LIN {X 0,Y 175.973,Z 623.597,A -85,B 0,C 180,E1 -22407.711,E2 -22407.711} C_VEL
LIN {X 0,Y 176.091,Z 624.209,A -85,B 0,C 180,E1 -22410,E2 -22410} C_VEL
LIN {X 0,Y 175.945,Z 624.405,A -85,B 0,C 180,E1 -22414.582,E2 -22414.582} C_VEL
LIN {X 0,Y 176.345,Z 623.273,A -85,B 0,C 180,E1 -22419.173,E2 -22419.173} C_VEL
LIN {X 0,Y 177.477,Z 620.803,A -85,B 0,C 180,E1 -22423.745,E2 -22423.745} C_VEL
LIN {X 0,Y 179.709,Z 616.939,A -85,B 0,C 180,E1 -22428.232,E2 -22428.232} C_VEL
LIN {X 0,Y 182.559,Z 611.727,A -85,B 0,C 180,E1 -22432.493,E2 -22432.493} C_VEL
LIN {X 0,Y 185.735,Z 606.375,A -85,B 0,C 180,E1 -22435.795,E2 -22435.795} C_VEL
LIN {X 0,Y 189.98,Z 599.018,A -85,B 0,C 180,E1 -22439.352,E2 -22439.352} C_VEL
LIN {X 0,Y 194.974,Z 589.893,A -85,B 0,C 180,E1 -22442.731,E2 -22442.731} C_VEL
LIN {X 0,Y 199.815,Z 580.368,A -85,B 0,C 180,E1 -22445.475,E2 -22445.475} C_VEL
LIN {X 0,Y 204.272,Z 570.439,A -85,B 0,C 180,E1 -22447.774,E2 -22447.774} C_VEL
LIN {X 0,Y 208.64,Z 559.5,A -85,B 0,C 180,E1 -22449.793,E2 -22449.793} C_VEL
LIN {X 0,Y 213.078,Z 546.888,A -85,B 0,C 180,E1 -22451.59,E2 -22451.59} C_VEL
LIN {X 0,Y 216.743,Z 534.645,A -85,B 0,C 180,E1 -22452.917,E2 -22452.917} C_VEL
LIN {X 0,Y 219.97,Z 521.133,A -85,B 0,C 180,E1 -22454.02,E2 -22454.02} C_VEL
LIN {X 0,Y 222.451,Z 506.848,A -85,B 0,C 180,E1 -22454.855,E2 -22454.855} C_VEL
LIN {X 0,Y 224.016,Z 492.183,A -85,B 0,C 180,E1 -22455.41,E2 -22455.41} C_VEL
LIN {X 0,Y 227.477,Z 439.874,A -85,B 0,C 180,E1 -22456.878,E2 -22456.878} C_VEL
LIN {X 0,Y 222.194,Z 427.229,A -85,B 0,C 180,E1 -22459.105,E2 -22459.105} C_VEL
LIN {X 0,Y 216.883,Z 416.225,A -85,B 0,C 180,E1 -22461.484,E2 -22461.484} C_VEL
LIN {X 0,Y 210.927,Z 405.095,A -85,B 0,C 180,E1 -22464.409,E2 -22464.409} C_VEL
LIN {X 0,Y 204.85,Z 394.973,A -85,B 0,C 180,E1 -22467.765,E2 -22467.765} C_VEL
LIN {X 0,Y 201.102,Z 389.341,A -85,B 0,C 180,E1 -22470.085,E2 -22470.085} C_VEL
LIN {X 0,Y 197.646,Z 384.334,A -85,B 0,C 180,E1 -22472.467,E2 -22472.467} C_VEL
LIN {X 0,Y 194.879,Z 381.371,A -85,B 0,C 180,E1 -22474.511,E2 -22474.511} C_VEL
LIN {X 0,Y 193.552,Z 379.243,A -85,B 0,C 180,E1 -22475.645,E2 -22475.645} C_VEL
LIN {X 0,Y 190.782,Z 376.698,A -85,B 0,C 180,E1 -22478.065,E2 -22478.065} C_VEL
LIN {X 0,Y 189.1,Z 373.76,A -85,B 0,C 180,E1 -22479.893,E2 -22479.893} C_VEL
LIN {X 0,Y 186.16,Z 371.606,A -85,B 0,C 180,E1 -22483.271,E2 -22483.271} C_VEL
LIN {X 0,Y 184.729,Z 369.094,A -85,B 0,C 180,E1 -22485.543,E2 -22485.543} C_VEL
LIN {X 0,Y 184.415,Z 367.934,A -85,B 0,C 180,E1 -22486.221,E2 -22486.221} C_VEL
LIN {X 0,Y 180.968,Z 365.75,A -85,B 0,C 180,E1 -22497.775,E2 -22497.775} C_VEL
LIN {X 0,Y 181.188,Z 365.794,A -85,B 0,C 180,E1 -22500.556,E2 -22500.556} C_VEL
LIN {X 0,Y 183.53,Z 367.618,A -85,B 0,C 180,E1 -22507.703,E2 -22507.703} C_VEL
LIN {X 0,Y 184.611,Z 368.106,A -85,B 0,C 180,E1 -22509.542,E2 -22509.542} C_VEL
LIN {X 0,Y 185.587,Z 370.744,A -85,B 0,C 180,E1 -22511.33,E2 -22511.33} C_VEL
LIN {X 0,Y 187.715,Z 373.002,A -85,B 0,C 180,E1 -22514.086,E2 -22514.086} C_VEL
LIN {X 0,Y 189.365,Z 373.966,A -85,B 0,C 180,E1 -22515.817,E2 -22515.817} C_VEL
LIN {X 0,Y 191.087,Z 377.097,A -85,B 0,C 180,E1 -22517.669,E2 -22517.669} C_VEL
LIN {X 0,Y 193.934,Z 379.745,A -85,B 0,C 180,E1 -22520.116,E2 -22520.116} C_VEL
LIN {X 0,Y 196.242,Z 383.109,A -85,B 0,C 180,E1 -22521.985,E2 -22521.985} C_VEL
LIN {X 0,Y 198.131,Z 385.043,A -85,B 0,C 180,E1 -22523.323,E2 -22523.323} C_VEL
LIN {X 0,Y 200.929,Z 388.709,A -85,B 0,C 180,E1 -22525.212,E2 -22525.212} C_VEL
LIN {X 0,Y 202.67,Z 391.076,A -85,B 0,C 180,E1 -22526.31,E2 -22526.31} C_VEL
LIN {X 0,Y 205.511,Z 394.828,A -85,B 0,C 180,E1 -22527.98,E2 -22527.98} C_VEL
LIN {X 0,Y 210.882,Z 402.349,A -85,B 0,C 180,E1 -22530.844,E2 -22530.844} C_VEL
LIN {X 0,Y 217.896,Z 413.285,A -85,B 0,C 180,E1 -22534.155,E2 -22534.155} C_VEL
LIN {X 0,Y 222.849,Z 422.031,A -85,B 0,C 180,E1 -22536.28,E2 -22536.28} C_VEL
LIN {X 0,Y 227.882,Z 432.924,A -85,B 0,C 180,E1 -22538.349,E2 -22538.349} C_VEL
LIN {X 0,Y 223.972,Z 490.841,A -85,B 0,C 180,E1 -22540.036,E2 -22540.036} C_VEL
LIN {X 0,Y 222.064,Z 505.188,A -85,B 0,C 180,E1 -22540.748,E2 -22540.748} C_VEL
LIN {X 0,Y 219.175,Z 519.704,A -85,B 0,C 180,E1 -22541.795,E2 -22541.795} C_VEL
LIN {X 0,Y 215.825,Z 532.368,A -85,B 0,C 180,E1 -22543.025,E2 -22543.025} C_VEL
LIN {X 0,Y 212.116,Z 544.319,A -85,B 0,C 180,E1 -22544.573,E2 -22544.573} C_VEL
LIN {X 0,Y 207.881,Z 555.831,A -85,B 0,C 180,E1 -22546.462,E2 -22546.462} C_VEL
LIN {X 0,Y 203.787,Z 565.394,A -85,B 0,C 180,E1 -22548.404,E2 -22548.404} C_VEL
LIN {X 0,Y 199.332,Z 575.034,A -85,B 0,C 180,E1 -22550.867,E2 -22550.867} C_VEL
LIN {X 0,Y 195.109,Z 583.394,A -85,B 0,C 180,E1 -22553.534,E2 -22553.534} C_VEL
LIN {X 0,Y 190.261,Z 591.993,A -85,B 0,C 180,E1 -22556.985,E2 -22556.985} C_VEL
LIN {X 0,Y 186.147,Z 598.901,A -85,B 0,C 180,E1 -22560.605,E2 -22560.605} C_VEL
LIN {X 0,Y 183.235,Z 603.656,A -85,B 0,C 180,E1 -22563.827,E2 -22563.827} C_VEL
LIN {X 0,Y 180.146,Z 608.557,A -85,B 0,C 180,E1 -22568.246,E2 -22568.246} C_VEL
LIN {X 0,Y 178.42,Z 611.225,A -85,B 0,C 180,E1 -22571.632,E2 -22571.632} C_VEL
LIN {X 0,Y 176.763,Z 613.538,A -85,B 0,C 180,E1 -22576.198,E2 -22576.198} C_VEL
LIN {X 0,Y 176.071,Z 614.498,A -85,B 0,C 180,E1 -22580.813,E2 -22580.813} C_VEL
LIN {X 0,Y 175.97,Z 614.139,A -85,B 0,C 180,E1 -22585.418,E2 -22585.418} C_VEL
LIN {X 0,Y 176.17,Z 612.472,A -85,B 0,C 180,E1 -22590,E2 -22590} C_VEL
LIN {X 0,Y 176.9,Z 609.462,A -85,B 0,C 180,E1 -22594.557,E2 -22594.557} C_VEL
LIN {X 0,Y 178.404,Z 605.021,A -85,B 0,C 180,E1 -22599.066,E2 -22599.066} C_VEL
LIN {X 0,Y 180.075,Z 600.613,A -85,B 0,C 180,E1 -22602.395,E2 -22602.395} C_VEL
LIN {X 0,Y 182.054,Z 595.264,A -85,B 0,C 180,E1 -22605.678,E2 -22605.678} C_VEL
LIN {X 0,Y 184.936,Z 587.607,A -85,B 0,C 180,E1 -22609.422,E2 -22609.422} C_VEL
LIN {X 0,Y 188.315,Z 579.592,A -85,B 0,C 180,E1 -22612.491,E2 -22612.491} C_VEL
LIN {X 0,Y 191.947,Z 569.95,A -85,B 0,C 180,E1 -22615.481,E2 -22615.481} C_VEL
LIN {X 0,Y 195.507,Z 559.268,A -85,B 0,C 180,E1 -22618.152,E2 -22618.152} C_VEL
LIN {X 0,Y 198.843,Z 548.7,A -85,B 0,C 180,E1 -22620.242,E2 -22620.242} C_VEL
LIN {X 0,Y 202.027,Z 537.334,A -85,B 0,C 180,E1 -22622.04,E2 -22622.04} C_VEL
LIN {X 0,Y 204.873,Z 525.038,A -85,B 0,C 180,E1 -22623.584,E2 -22623.584} C_VEL
LIN {X 0,Y 207.454,Z 511.398,A -85,B 0,C 180,E1 -22624.868,E2 -22624.868} C_VEL
LIN {X 0,Y 209.362,Z 497.206,A -85,B 0,C 180,E1 -22625.828,E2 -22625.828} C_VEL
LIN {X 0,Y 210.555,Z 483.575,A -85,B 0,C 180,E1 -22626.407,E2 -22626.407} C_VEL
LIN {X 0,Y 214.132,Z 420.681,A -85,B 0,C 180,E1 -22628.327,E2 -22628.327} C_VEL
LIN {X 0,Y 209.725,Z 410.077,A -85,B 0,C 180,E1 -22629.873,E2 -22629.873} C_VEL
LIN {X 0,Y 202.836,Z 397.568,A -85,B 0,C 180,E1 -22632.31,E2 -22632.31} C_VEL
LIN {X 0,Y 195.932,Z 386.643,A -85,B 0,C 180,E1 -22634.959,E2 -22634.959} C_VEL
LIN {X 0,Y 191.272,Z 379.912,A -85,B 0,C 180,E1 -22636.904,E2 -22636.904} C_VEL
LIN {X 0,Y 188.461,Z 376.039,A -85,B 0,C 180,E1 -22638.153,E2 -22638.153} C_VEL
LIN {X 0,Y 185.501,Z 371.965,A -85,B 0,C 180,E1 -22639.547,E2 -22639.547} C_VEL
LIN {X 0,Y 183.117,Z 369.127,A -85,B 0,C 180,E1 -22640.708,E2 -22640.708} C_VEL
LIN {X 0,Y 182.006,Z 367.177,A -85,B 0,C 180,E1 -22641.312,E2 -22641.312} C_VEL
LIN {X 0,Y 179.721,Z 365.124,A -85,B 0,C 180,E1 -22642.472,E2 -22642.472} C_VEL
LIN {X 0,Y 178.594,Z 362.743,A -85,B 0,C 180,E1 -22643.165,E2 -22643.165} C_VEL
LIN {X 0,Y 178.432,Z 361.874,A -85,B 0,C 180,E1 -22643.38,E2 -22643.38} C_VEL
LIN {X 0,Y 178.486,Z 361.865,A -85,B 0,C 180,E1 -22646.546,E2 -22646.546} C_VEL
LIN {X 0,Y 178.441,Z 361.868,A -85,B 0,C 180,E1 -22651.794,E2 -22651.794} C_VEL
LIN {X 0,Y 178.507,Z 361.874,A -85,B 0,C 180,E1 -22654.896,E2 -22654.896} C_VEL
LIN {X 0,Y 178.608,Z 361.83,A -85,B 0,C 180,E1 -22661.651,E2 -22661.651} C_VEL
LIN {X 0,Y 178.636,Z 361.834,A -85,B 0,C 180,E1 -22666.345,E2 -22666.345} C_VEL
LIN {X 0,Y 178.908,Z 361.788,A -85,B 0,C 180,E1 -22670.959,E2 -22670.959} C_VEL
LIN {X 0,Y 179.145,Z 361.792,A -85,B 0,C 180,E1 -22677.751,E2 -22677.751} C_VEL
LIN {X 0,Y 179.348,Z 361.762,A -85,B 0,C 180,E1 -22679.999,E2 -22679.999} C_VEL
LIN {X 0,Y 178.84,Z 361.827,A -85,B 0,C 180,E1 -22684.507,E2 -22684.507} C_VEL
LIN {X 0,Y 178.908,Z 361.819,A -85,B 0,C 180,E1 -22689.04,E2 -22689.04} C_VEL
LIN {X 0,Y 178.661,Z 361.848,A -85,B 0,C 180,E1 -22693.651,E2 -22693.651} C_VEL
LIN {X 0,Y 178.624,Z 361.855,A -85,B 0,C 180,E1 -22699.215,E2 -22699.215} C_VEL
LIN {X 0,Y 178.52,Z 361.869,A -85,B 0,C 180,E1 -22705.113,E2 -22705.113} C_VEL
LIN {X 0,Y 178.464,Z 361.884,A -85,B 0,C 180,E1 -22710.793,E2 -22710.793} C_VEL
LIN {X 0,Y 178.485,Z 361.939,A -85,B 0,C 180,E1 -22711.365,E2 -22711.365} C_VEL
LIN {X 0,Y 179.333,Z 364.467,A -85,B 0,C 180,E1 -22711.941,E2 -22711.941} C_VEL
LIN {X 0,Y 181.332,Z 366.723,A -85,B 0,C 180,E1 -22713,E2 -22713} C_VEL
LIN {X 0,Y 182.467,Z 367.748,A -85,B 0,C 180,E1 -22713.563,E2 -22713.563} C_VEL
LIN {X 0,Y 184.533,Z 370.957,A -85,B 0,C 180,E1 -22714.636,E2 -22714.636} C_VEL
LIN {X 0,Y 186.21,Z 372.706,A -85,B 0,C 180,E1 -22715.418,E2 -22715.418} C_VEL
LIN {X 0,Y 188.828,Z 376.357,A -85,B 0,C 180,E1 -22716.641,E2 -22716.641} C_VEL
LIN {X 0,Y 194.381,Z 385.325,A -85,B 0,C 180,E1 -22719.1,E2 -22719.1} C_VEL
LIN {X 0,Y 201.137,Z 397.747,A -85,B 0,C 180,E1 -22721.848,E2 -22721.848} C_VEL
LIN {X 0,Y 206.577,Z 409.402,A -85,B 0,C 180,E1 -22723.922,E2 -22723.922} C_VEL
LIN {X 0,Y 211.631,Z 421.789,A -85,B 0,C 180,E1 -22725.765,E2 -22725.765} C_VEL
LIN {X 0,Y 213.853,Z 427.885,A -85,B 0,C 180,E1 -22726.56,E2 -22726.56} C_VEL
LIN {X 0,Y 212.024,Z 460.209,A -85,B 0,C 180,E1 -22727.546,E2 -22727.546} C_VEL
LIN {X 0,Y 211.141,Z 466.055,A -85,B 0,C 180,E1 -22727.599,E2 -22727.599} C_VEL
LIN {X 0,Y 205.631,Z 485.05,A -85,B 0,C 180,E1 -22727.161,E2 -22727.161} C_VEL
LIN {X 0,Y 204.839,Z 490.89,A -85,B 0,C 180,E1 -22727.236,E2 -22727.236} C_VEL
LIN {X 0,Y 203.51,Z 505.696,A -85,B 0,C 180,E1 -22727.836,E2 -22727.836} C_VEL
LIN {X 0,Y 201.524,Z 518.899,A -85,B 0,C 180,E1 -22728.667,E2 -22728.667} C_VEL
LIN {X 0,Y 198.648,Z 533.064,A -85,B 0,C 180,E1 -22729.949,E2 -22729.949} C_VEL
LIN {X 0,Y 195.227,Z 546.537,A -85,B 0,C 180,E1 -22731.612,E2 -22731.612} C_VEL
LIN {X 0,Y 191.793,Z 558.043,A -85,B 0,C 180,E1 -22733.454,E2 -22733.454} C_VEL
LIN {X 0,Y 187.889,Z 569.824,A -85,B 0,C 180,E1 -22735.87,E2 -22735.87} C_VEL
LIN {X 0,Y 184.218,Z 579.566,A -85,B 0,C 180,E1 -22738.361,E2 -22738.361} C_VEL
LIN {X 0,Y 180.311,Z 589.317,A -85,B 0,C 180,E1 -22741.48,E2 -22741.48} C_VEL
LIN {X 0,Y 177.019,Z 597.403,A -85,B 0,C 180,E1 -22744.736,E2 -22744.736} C_VEL
LIN {X 0,Y 173.979,Z 605.158,A -85,B 0,C 180,E1 -22748.681,E2 -22748.681} C_VEL
LIN {X 0,Y 171.98,Z 610.552,A -85,B 0,C 180,E1 -22752.152,E2 -22752.152} C_VEL
LIN {X 0,Y 170.042,Z 616.224,A -85,B 0,C 180,E1 -22756.861,E2 -22756.861} C_VEL
LIN {X 0,Y 169.291,Z 619.418,A -85,B 0,C 180,E1 -22760.441,E2 -22760.441} C_VEL
LIN {X 0,Y 168.872,Z 622.398,A -85,B 0,C 180,E1 -22765.226,E2 -22765.226} C_VEL
LIN {X 0,Y 168.999,Z 623.988,A -85,B 0,C 180,E1 -22770,E2 -22770} C_VEL
LIN {X 0,Y 168.858,Z 624.209,A -85,B 0,C 180,E1 -22774.775,E2 -22774.775} C_VEL
LIN {X 0,Y 169.313,Z 623.103,A -85,B 0,C 180,E1 -22779.558,E2 -22779.558} C_VEL
LIN {X 0,Y 170.54,Z 620.658,A -85,B 0,C 180,E1 -22784.316,E2 -22784.316} C_VEL
LIN {X 0,Y 172.915,Z 616.823,A -85,B 0,C 180,E1 -22788.975,E2 -22788.975} C_VEL
LIN {X 0,Y 175.71,Z 612.052,A -85,B 0,C 180,E1 -22793.083,E2 -22793.083} C_VEL
LIN {X 0,Y 179.33,Z 606.318,A -85,B 0,C 180,E1 -22796.788,E2 -22796.788} C_VEL
LIN {X 0,Y 183.82,Z 598.996,A -85,B 0,C 180,E1 -22800.437,E2 -22800.437} C_VEL
LIN {X 0,Y 189.023,Z 589.929,A -85,B 0,C 180,E1 -22803.898,E2 -22803.898} C_VEL
LIN {X 0,Y 194.063,Z 580.452,A -85,B 0,C 180,E1 -22806.695,E2 -22806.695} C_VEL
LIN {X 0,Y 198.977,Z 569.923,A -85,B 0,C 180,E1 -22809.166,E2 -22809.166} C_VEL
LIN {X 0,Y 203.729,Z 558.427,A -85,B 0,C 180,E1 -22811.281,E2 -22811.281} C_VEL
LIN {X 0,Y 208.356,Z 545.62,A -85,B 0,C 180,E1 -22813.083,E2 -22813.083} C_VEL
LIN {X 0,Y 212.154,Z 533.106,A -85,B 0,C 180,E1 -22814.412,E2 -22814.412} C_VEL
LIN {X 0,Y 215.482,Z 519.186,A -85,B 0,C 180,E1 -22815.517,E2 -22815.517} C_VEL
LIN {X 0,Y 217.93,Z 505.007,A -85,B 0,C 180,E1 -22816.308,E2 -22816.308} C_VEL
LIN {X 0,Y 219.421,Z 490.456,A -85,B 0,C 180,E1 -22816.823,E2 -22816.823} C_VEL
LIN {X 0,Y 222.682,Z 442.18,A -85,B 0,C 180,E1 -22818.203,E2 -22818.203} C_VEL
LIN {X 0,Y 217.268,Z 429.212,A -85,B 0,C 180,E1 -22820.645,E2 -22820.645} C_VEL
LIN {X 0,Y 211.876,Z 418.079,A -85,B 0,C 180,E1 -22823.255,E2 -22823.255} C_VEL
LIN {X 0,Y 206.958,Z 409.008,A -85,B 0,C 180,E1 -22825.858,E2 -22825.858} C_VEL
LIN {X 0,Y 202.253,Z 400.832,A -85,B 0,C 180,E1 -22828.64,E2 -22828.64} C_VEL
LIN {X 0,Y 198.512,Z 395.039,A -85,B 0,C 180,E1 -22831.088,E2 -22831.088} C_VEL
LIN {X 0,Y 195.64,Z 390.778,A -85,B 0,C 180,E1 -22833.174,E2 -22833.174} C_VEL
LIN {X 0,Y 192.819,Z 387.498,A -85,B 0,C 180,E1 -22835.383,E2 -22835.383} C_VEL
LIN {X 0,Y 191.719,Z 385.818,A -85,B 0,C 180,E1 -22836.362,E2 -22836.362} C_VEL
LIN {X 0,Y 188.944,Z 382.931,A -85,B 0,C 180,E1 -22838.951,E2 -22838.951} C_VEL
LIN {X 0,Y 187.765,Z 380.683,A -85,B 0,C 180,E1 -22840.314,E2 -22840.314} C_VEL
LIN {X 0,Y 184.681,Z 378.12,A -85,B 0,C 180,E1 -22844.074,E2 -22844.074} C_VEL
LIN {X 0,Y 183.29,Z 375.312,A -85,B 0,C 180,E1 -22846.532,E2 -22846.532} C_VEL
LIN {X 0,Y 182.918,Z 374.828,A -85,B 0,C 180,E1 -22847.237,E2 -22847.237} C_VEL
LIN {X 0,Y 180.109,Z 373.009,A -85,B 0,C 180,E1 -22856.645,E2 -22856.645} C_VEL
LIN {X 0,Y 180.319,Z 372.862,A -85,B 0,C 180,E1 -22860.559,E2 -22860.559} C_VEL
LIN {X 0,Y 183.365,Z 375.104,A -85,B 0,C 180,E1 -22868.983,E2 -22868.983} C_VEL
LIN {X 0,Y 184.611,Z 377.969,A -85,B 0,C 180,E1 -22871.252,E2 -22871.252} C_VEL
LIN {X 0,Y 187.098,Z 380.28,A -85,B 0,C 180,E1 -22874.411,E2 -22874.411} C_VEL
LIN {X 0,Y 187.967,Z 381.046,A -85,B 0,C 180,E1 -22875.363,E2 -22875.363} C_VEL
LIN {X 0,Y 190.004,Z 384.344,A -85,B 0,C 180,E1 -22877.557,E2 -22877.557} C_VEL
LIN {X 0,Y 192.192,Z 386.43,A -85,B 0,C 180,E1 -22879.493,E2 -22879.493} C_VEL
LIN {X 0,Y 194.857,Z 390.099,A -85,B 0,C 180,E1 -22881.697,E2 -22881.697} C_VEL
LIN {X 0,Y 196.224,Z 391.657,A -85,B 0,C 180,E1 -22882.707,E2 -22882.707} C_VEL
LIN {X 0,Y 199.87,Z 396.488,A -85,B 0,C 180,E1 -22885.222,E2 -22885.222} C_VEL
LIN {X 0,Y 203.179,Z 401.084,A -85,B 0,C 180,E1 -22887.279,E2 -22887.279} C_VEL
LIN {X 0,Y 208.123,Z 408.223,A -85,B 0,C 180,E1 -22890.04,E2 -22890.04} C_VEL
LIN {X 0,Y 214.742,Z 418.833,A -85,B 0,C 180,E1 -22893.318,E2 -22893.318} C_VEL
LIN {X 0,Y 219.279,Z 427.096,A -85,B 0,C 180,E1 -22895.368,E2 -22895.368} C_VEL
LIN {X 0,Y 223.12,Z 435.581,A -85,B 0,C 180,E1 -22897.044,E2 -22897.044} C_VEL
LIN {X 0,Y 219.269,Z 490.617,A -85,B 0,C 180,E1 -22898.654,E2 -22898.654} C_VEL
LIN {X 0,Y 217.323,Z 505.011,A -85,B 0,C 180,E1 -22899.366,E2 -22899.366} C_VEL
LIN {X 0,Y 214.465,Z 519.054,A -85,B 0,C 180,E1 -22900.367,E2 -22900.367} C_VEL
LIN {X 0,Y 211,Z 531.905,A -85,B 0,C 180,E1 -22901.602,E2 -22901.602} C_VEL
LIN {X 0,Y 207.625,Z 542.648,A -85,B 0,C 180,E1 -22902.97,E2 -22902.97} C_VEL
LIN {X 0,Y 203.221,Z 554.41,A -85,B 0,C 180,E1 -22904.85,E2 -22904.85} C_VEL
LIN {X 0,Y 198.434,Z 565.226,A -85,B 0,C 180,E1 -22907.016,E2 -22907.016} C_VEL
LIN {X 0,Y 193.433,Z 575.643,A -85,B 0,C 180,E1 -22909.73,E2 -22909.73} C_VEL
LIN {X 0,Y 188.601,Z 584.697,A -85,B 0,C 180,E1 -22912.732,E2 -22912.732} C_VEL
LIN {X 0,Y 183.578,Z 593.102,A -85,B 0,C 180,E1 -22916.281,E2 -22916.281} C_VEL
LIN {X 0,Y 179.903,Z 598.932,A -85,B 0,C 180,E1 -22919.479,E2 -22919.479} C_VEL
LIN {X 0,Y 176.78,Z 603.724,A -85,B 0,C 180,E1 -22922.794,E2 -22922.794} C_VEL
LIN {X 0,Y 173.478,Z 608.659,A -85,B 0,C 180,E1 -22927.364,E2 -22927.364} C_VEL
LIN {X 0,Y 171.594,Z 611.36,A -85,B 0,C 180,E1 -22930.873,E2 -22930.873} C_VEL
LIN {X 0,Y 169.81,Z 613.703,A -85,B 0,C 180,E1 -22935.621,E2 -22935.621} C_VEL
LIN {X 0,Y 169.013,Z 614.694,A -85,B 0,C 180,E1 -22940.425,E2 -22940.425} C_VEL
LIN {X 0,Y 168.869,Z 614.364,A -85,B 0,C 180,E1 -22945.225,E2 -22945.225} C_VEL
LIN {X 0,Y 168.95,Z 613.709,A -85,B 0,C 180,E1 -22947.616,E2 -22947.616} C_VEL
LIN {X 0,Y 169.379,Z 611.408,A -85,B 0,C 180,E1 -22952.378,E2 -22952.378} C_VEL
LIN {X 0,Y 170.498,Z 607.73,A -85,B 0,C 180,E1 -22957.103,E2 -22957.103} C_VEL
LIN {X 0,Y 172.547,Z 602.553,A -85,B 0,C 180,E1 -22961.751,E2 -22961.751} C_VEL
LIN {X 0,Y 174.504,Z 597.539,A -85,B 0,C 180,E1 -22965.176,E2 -22965.176} C_VEL
LIN {X 0,Y 177.311,Z 590.395,A -85,B 0,C 180,E1 -22969.087,E2 -22969.087} C_VEL
LIN {X 0,Y 180.54,Z 582.895,A -85,B 0,C 180,E1 -22972.305,E2 -22972.305} C_VEL
LIN {X 0,Y 184.293,Z 573.891,A -85,B 0,C 180,E1 -22975.405,E2 -22975.405} C_VEL
LIN {X 0,Y 188.282,Z 563.014,A -85,B 0,C 180,E1 -22978.419,E2 -22978.419} C_VEL
LIN {X 0,Y 191.914,Z 551.949,A -85,B 0,C 180,E1 -22980.843,E2 -22980.843} C_VEL
LIN {X 0,Y 195.183,Z 541.209,A -85,B 0,C 180,E1 -22982.691,E2 -22982.691} C_VEL
LIN {X 0,Y 198.59,Z 527.96,A -85,B 0,C 180,E1 -22984.488,E2 -22984.488} C_VEL
LIN {X 0,Y 201.268,Z 515.158,A -85,B 0,C 180,E1 -22985.795,E2 -22985.795} C_VEL
LIN {X 0,Y 203.501,Z 500.59,A -85,B 0,C 180,E1 -22986.874,E2 -22986.874} C_VEL
LIN {X 0,Y 204.807,Z 487.533,A -85,B 0,C 180,E1 -22987.524,E2 -22987.524} C_VEL
LIN {X 0,Y 208.747,Z 422.815,A -85,B 0,C 180,E1 -22989.536,E2 -22989.536} C_VEL
LIN {X 0,Y 204.973,Z 413.798,A -85,B 0,C 180,E1 -22990.935,E2 -22990.935} C_VEL
LIN {X 0,Y 198.773,Z 402.384,A -85,B 0,C 180,E1 -22993.253,E2 -22993.253} C_VEL
LIN {X 0,Y 192.357,Z 392.011,A -85,B 0,C 180,E1 -22995.849,E2 -22995.849} C_VEL
LIN {X 0,Y 186.842,Z 383.9,A -85,B 0,C 180,E1 -22998.295,E2 -22998.295} C_VEL
LIN {X 0,Y 182.307,Z 377.673,A -85,B 0,C 180,E1 -23000.497,E2 -23000.497} C_VEL
LIN {X 0,Y 179.696,Z 374.172,A -85,B 0,C 180,E1 -23001.866,E2 -23001.866} C_VEL
LIN {X 0,Y 178.672,Z 372.913,A -85,B 0,C 180,E1 -23002.419,E2 -23002.419} C_VEL
LIN {X 0,Y 176.34,Z 370.094,A -85,B 0,C 180,E1 -23003.729,E2 -23003.729} C_VEL
LIN {X 0,Y 175.434,Z 368.318,A -85,B 0,C 180,E1 -23004.31,E2 -23004.31} C_VEL
LIN {X 0,Y 173.084,Z 366.459,A -85,B 0,C 180,E1 -23005.678,E2 -23005.678} C_VEL
LIN {X 0,Y 171.709,Z 363.987,A -85,B 0,C 180,E1 -23006.633,E2 -23006.633} C_VEL
LIN {X 0,Y 171.434,Z 362.741,A -85,B 0,C 180,E1 -23006.923,E2 -23006.923} C_VEL
LIN {X 0,Y 171.41,Z 362.755,A -85,B 0,C 180,E1 -23010.526,E2 -23010.526} C_VEL
LIN {X 0,Y 171.429,Z 362.755,A -85,B 0,C 180,E1 -23015.796,E2 -23015.796} C_VEL
LIN {X 0,Y 171.509,Z 362.706,A -85,B 0,C 180,E1 -23020.863,E2 -23020.863} C_VEL
LIN {X 0,Y 171.551,Z 362.726,A -85,B 0,C 180,E1 -23025.77,E2 -23025.77} C_VEL
LIN {X 0,Y 171.846,Z 362.662,A -85,B 0,C 180,E1 -23030.584,E2 -23030.584} C_VEL
LIN {X 0,Y 171.8,Z 362.702,A -85,B 0,C 180,E1 -23035.306,E2 -23035.306} C_VEL
LIN {X 0,Y 172.313,Z 362.638,A -85,B 0,C 180,E1 -23039.999,E2 -23039.999} C_VEL
LIN {X 0,Y 171.789,Z 362.704,A -85,B 0,C 180,E1 -23044.693,E2 -23044.693} C_VEL
LIN {X 0,Y 171.846,Z 362.696,A -85,B 0,C 180,E1 -23049.415,E2 -23049.415} C_VEL
LIN {X 0,Y 171.578,Z 362.729,A -85,B 0,C 180,E1 -23054.226,E2 -23054.226} C_VEL
LIN {X 0,Y 171.543,Z 362.739,A -85,B 0,C 180,E1 -23059.559,E2 -23059.559} C_VEL
LIN {X 0,Y 171.458,Z 362.747,A -85,B 0,C 180,E1 -23065.607,E2 -23065.607} C_VEL
LIN {X 0,Y 171.417,Z 362.761,A -85,B 0,C 180,E1 -23067.715,E2 -23067.715} C_VEL
LIN {X 0,Y 172.229,Z 365.264,A -85,B 0,C 180,E1 -23068.401,E2 -23068.401} C_VEL
LIN {X 0,Y 174.163,Z 367.52,A -85,B 0,C 180,E1 -23069.616,E2 -23069.616} C_VEL
LIN {X 0,Y 175.634,Z 368.577,A -85,B 0,C 180,E1 -23070.449,E2 -23070.449} C_VEL
LIN {X 0,Y 177.573,Z 371.807,A -85,B 0,C 180,E1 -23071.628,E2 -23071.628} C_VEL
LIN {X 0,Y 179.61,Z 373.911,A -85,B 0,C 180,E1 -23072.715,E2 -23072.715} C_VEL
LIN {X 0,Y 182.208,Z 377.474,A -85,B 0,C 180,E1 -23074.085,E2 -23074.085} C_VEL
LIN {X 0,Y 183.769,Z 379.597,A -85,B 0,C 180,E1 -23074.869,E2 -23074.869} C_VEL
LIN {X 0,Y 186.521,Z 383.401,A -85,B 0,C 180,E1 -23076.191,E2 -23076.191} C_VEL
LIN {X 0,Y 192.036,Z 392.933,A -85,B 0,C 180,E1 -23078.732,E2 -23078.732} C_VEL
LIN {X 0,Y 197.835,Z 404.088,A -85,B 0,C 180,E1 -23081.189,E2 -23081.189} C_VEL
LIN {X 0,Y 203.199,Z 416.067,A -85,B 0,C 180,E1 -23083.331,E2 -23083.331} C_VEL
LIN {X 0,Y 208.436,Z 429.77,A -85,B 0,C 180,E1 -23085.341,E2 -23085.341} C_VEL
LIN {X 0,Y 204.839,Z 490.89,A -85,B 0,C 180,E1 -23087.236,E2 -23087.236} C_VEL
LIN {X 0,Y 203.962,Z 496.72,A -85,B 0,C 180,E1 -23087.323,E2 -23087.323} C_VEL
LIN {X 0,Y 200.776,Z 506.11,A -85,B 0,C 180,E1 -23087.227,E2 -23087.227} C_VEL
LIN {X 0,Y 197.16,Z 515.362,A -85,B 0,C 180,E1 -23087.247,E2 -23087.247} C_VEL
LIN {X 0,Y 195.628,Z 520.979,A -85,B 0,C 180,E1 -23087.548,E2 -23087.548} C_VEL
LIN {X 0,Y 192.562,Z 535.224,A -85,B 0,C 180,E1 -23088.932,E2 -23088.932} C_VEL
LIN {X 0,Y 189.216,Z 547.414,A -85,B 0,C 180,E1 -23090.501,E2 -23090.501} C_VEL
LIN {X 0,Y 185.686,Z 558.726,A -85,B 0,C 180,E1 -23092.388,E2 -23092.388} C_VEL
LIN {X 0,Y 181.618,Z 570.354,A -85,B 0,C 180,E1 -23094.857,E2 -23094.857} C_VEL
LIN {X 0,Y 177.459,Z 580.874,A -85,B 0,C 180,E1 -23097.68,E2 -23097.68} C_VEL
LIN {X 0,Y 173.429,Z 590.371,A -85,B 0,C 180,E1 -23100.903,E2 -23100.903} C_VEL
LIN {X 0,Y 169.505,Z 599.409,A -85,B 0,C 180,E1 -23104.85,E2 -23104.85} C_VEL
LIN {X 0,Y 166.585,Z 606.722,A -85,B 0,C 180,E1 -23108.985,E2 -23108.985} C_VEL
LIN {X 0,Y 164.552,Z 611.834,A -85,B 0,C 180,E1 -23112.604,E2 -23112.604} C_VEL
LIN {X 0,Y 162.742,Z 617.095,A -85,B 0,C 180,E1 -23117.53,E2 -23117.53} C_VEL
LIN {X 0,Y 161.926,Z 620.825,A -85,B 0,C 180,E1 -23122.518,E2 -23122.518} C_VEL
LIN {X 0,Y 161.795,Z 623.13,A -85,B 0,C 180,E1 -23127.511,E2 -23127.511} C_VEL
LIN {X 0,Y 161.91,Z 623.768,A -85,B 0,C 180,E1 -23130,E2 -23130} C_VEL
LIN {X 0,Y 161.795,Z 624.058,A -85,B 0,C 180,E1 -23132.49,E2 -23132.49} C_VEL
LIN {X 0,Y 161.931,Z 623.638,A -85,B 0,C 180,E1 -23137.481,E2 -23137.481} C_VEL
LIN {X 0,Y 162.837,Z 621.892,A -85,B 0,C 180,E1 -23142.463,E2 -23142.463} C_VEL
LIN {X 0,Y 164.784,Z 618.79,A -85,B 0,C 180,E1 -23147.371,E2 -23147.371} C_VEL
LIN {X 0,Y 167.804,Z 614.246,A -85,B 0,C 180,E1 -23152.144,E2 -23152.144} C_VEL
LIN {X 0,Y 170.66,Z 609.759,A -85,B 0,C 180,E1 -23155.621,E2 -23155.621} C_VEL
LIN {X 0,Y 174.896,Z 603.315,A -85,B 0,C 180,E1 -23159.489,E2 -23159.489} C_VEL
LIN {X 0,Y 179.916,Z 595.332,A -85,B 0,C 180,E1 -23163.153,E2 -23163.153} C_VEL
LIN {X 0,Y 184.874,Z 586.998,A -85,B 0,C 180,E1 -23166.103,E2 -23166.103} C_VEL
LIN {X 0,Y 190.191,Z 576.981,A -85,B 0,C 180,E1 -23168.917,E2 -23168.917} C_VEL
LIN {X 0,Y 195.435,Z 565.834,A -85,B 0,C 180,E1 -23171.36,E2 -23171.36} C_VEL
LIN {X 0,Y 200.578,Z 553.348,A -85,B 0,C 180,E1 -23173.444,E2 -23173.444} C_VEL
LIN {X 0,Y 204.899,Z 540.978,A -85,B 0,C 180,E1 -23175.027,E2 -23175.027} C_VEL
LIN {X 0,Y 208.903,Z 527.173,A -85,B 0,C 180,E1 -23176.329,E2 -23176.329} C_VEL
LIN {X 0,Y 211.94,Z 512.966,A -85,B 0,C 180,E1 -23177.325,E2 -23177.325} C_VEL
LIN {X 0,Y 214.093,Z 498.52,A -85,B 0,C 180,E1 -23177.995,E2 -23177.995} C_VEL
LIN {X 0,Y 218.051,Z 444.716,A -85,B 0,C 180,E1 -23179.561,E2 -23179.561} C_VEL
LIN {X 0,Y 213.103,Z 432.727,A -85,B 0,C 180,E1 -23181.946,E2 -23181.946} C_VEL
LIN {X 0,Y 208.23,Z 422.436,A -85,B 0,C 180,E1 -23184.468,E2 -23184.468} C_VEL
LIN {X 0,Y 203.699,Z 413.863,A -85,B 0,C 180,E1 -23187.029,E2 -23187.029} C_VEL
LIN {X 0,Y 199.512,Z 406.386,A -85,B 0,C 180,E1 -23189.663,E2 -23189.663} C_VEL
LIN {X 0,Y 196.154,Z 400.987,A -85,B 0,C 180,E1 -23191.995,E2 -23191.995} C_VEL
LIN {X 0,Y 193.526,Z 397.066,A -85,B 0,C 180,E1 -23194.003,E2 -23194.003} C_VEL
LIN {X 0,Y 190.605,Z 393.27,A -85,B 0,C 180,E1 -23196.461,E2 -23196.461} C_VEL
LIN {X 0,Y 189.79,Z 392.257,A -85,B 0,C 180,E1 -23197.208,E2 -23197.208} C_VEL
LIN {X 0,Y 187.171,Z 389.143,A -85,B 0,C 180,E1 -23199.838,E2 -23199.838} C_VEL
LIN {X 0,Y 186.107,Z 387.331,A -85,B 0,C 180,E1 -23201.116,E2 -23201.116} C_VEL
LIN {X 0,Y 183.345,Z 384.777,A -85,B 0,C 180,E1 -23204.721,E2 -23204.721} C_VEL
LIN {X 0,Y 181.918,Z 381.839,A -85,B 0,C 180,E1 -23207.45,E2 -23207.45} C_VEL
LIN {X 0,Y 179.236,Z 379.844,A -85,B 0,C 180,E1 -23217.753,E2 -23217.753} C_VEL
LIN {X 0,Y 179.45,Z 379.929,A -85,B 0,C 180,E1 -23220.562,E2 -23220.562} C_VEL
LIN {X 0,Y 182.172,Z 382.036,A -85,B 0,C 180,E1 -23228.459,E2 -23228.459} C_VEL
LIN {X 0,Y 183.458,Z 384.892,A -85,B 0,C 180,E1 -23230.887,E2 -23230.887} C_VEL
LIN {X 0,Y 185.781,Z 387.125,A -85,B 0,C 180,E1 -23233.956,E2 -23233.956} C_VEL
LIN {X 0,Y 186.516,Z 387.862,A -85,B 0,C 180,E1 -23234.805,E2 -23234.805} C_VEL
LIN {X 0,Y 188.524,Z 391.083,A -85,B 0,C 180,E1 -23237.048,E2 -23237.048} C_VEL
LIN {X 0,Y 190.463,Z 393.019,A -85,B 0,C 180,E1 -23238.841,E2 -23238.841} C_VEL
LIN {X 0,Y 193.184,Z 396.764,A -85,B 0,C 180,E1 -23241.177,E2 -23241.177} C_VEL
LIN {X 0,Y 194.374,Z 398.296,A -85,B 0,C 180,E1 -23242.103,E2 -23242.103} C_VEL
LIN {X 0,Y 197.86,Z 403.042,A -85,B 0,C 180,E1 -23244.607,E2 -23244.607} C_VEL
LIN {X 0,Y 201.101,Z 407.721,A -85,B 0,C 180,E1 -23246.705,E2 -23246.705} C_VEL
LIN {X 0,Y 205.366,Z 413.98,A -85,B 0,C 180,E1 -23249.188,E2 -23249.188} C_VEL
LIN {X 0,Y 211.796,Z 424.661,A -85,B 0,C 180,E1 -23252.535,E2 -23252.535} C_VEL
LIN {X 0,Y 215.618,Z 431.82,A -85,B 0,C 180,E1 -23254.354,E2 -23254.354} C_VEL
LIN {X 0,Y 218.453,Z 438.177,A -85,B 0,C 180,E1 -23255.67,E2 -23255.67} C_VEL
LIN {X 0,Y 214.62,Z 491.187,A -85,B 0,C 180,E1 -23257.25,E2 -23257.25} C_VEL
LIN {X 0,Y 212.577,Z 505.602,A -85,B 0,C 180,E1 -23257.973,E2 -23257.973} C_VEL
LIN {X 0,Y 209.63,Z 519.545,A -85,B 0,C 180,E1 -23258.978,E2 -23258.978} C_VEL
LIN {X 0,Y 205.828,Z 533.045,A -85,B 0,C 180,E1 -23260.296,E2 -23260.296} C_VEL
LIN {X 0,Y 202.102,Z 544.226,A -85,B 0,C 180,E1 -23261.762,E2 -23261.762} C_VEL
LIN {X 0,Y 197.197,Z 556.53,A -85,B 0,C 180,E1 -23263.804,E2 -23263.804} C_VEL
LIN {X 0,Y 192.319,Z 567.023,A -85,B 0,C 180,E1 -23266.026,E2 -23266.026} C_VEL
LIN {X 0,Y 187.002,Z 577.474,A -85,B 0,C 180,E1 -23268.892,E2 -23268.892} C_VEL
LIN {X 0,Y 182.108,Z 585.999,A -85,B 0,C 180,E1 -23271.867,E2 -23271.867} C_VEL
LIN {X 0,Y 176.931,Z 594.152,A -85,B 0,C 180,E1 -23275.526,E2 -23275.526} C_VEL
LIN {X 0,Y 172.548,Z 600.694,A -85,B 0,C 180,E1 -23279.394,E2 -23279.394} C_VEL
LIN {X 0,Y 168.47,Z 606.475,A -85,B 0,C 180,E1 -23284.022,E2 -23284.022} C_VEL
LIN {X 0,Y 166.123,Z 609.782,A -85,B 0,C 180,E1 -23287.619,E2 -23287.619} C_VEL
LIN {X 0,Y 163.719,Z 612.854,A -85,B 0,C 180,E1 -23292.513,E2 -23292.513} C_VEL
LIN {X 0,Y 162.287,Z 614.546,A -85,B 0,C 180,E1 -23297.495,E2 -23297.495} C_VEL
LIN {X 0,Y 161.813,Z 614.903,A -85,B 0,C 180,E1 -23302.513,E2 -23302.513} C_VEL
LIN {X 0,Y 161.844,Z 613.948,A -85,B 0,C 180,E1 -23307.511,E2 -23307.511} C_VEL
LIN {X 0,Y 162.291,Z 611.678,A -85,B 0,C 180,E1 -23312.482,E2 -23312.482} C_VEL
LIN {X 0,Y 163.464,Z 608.031,A -85,B 0,C 180,E1 -23317.411,E2 -23317.411} C_VEL
LIN {X 0,Y 165.611,Z 602.892,A -85,B 0,C 180,E1 -23322.25,E2 -23322.25} C_VEL
LIN {X 0,Y 167.671,Z 597.911,A -85,B 0,C 180,E1 -23325.81,E2 -23325.81} C_VEL
LIN {X 0,Y 170.645,Z 590.805,A -85,B 0,C 180,E1 -23329.863,E2 -23329.863} C_VEL
LIN {X 0,Y 174.028,Z 583.35,A -85,B 0,C 180,E1 -23333.188,E2 -23333.188} C_VEL
LIN {X 0,Y 177.94,Z 574.397,A -85,B 0,C 180,E1 -23336.381,E2 -23336.381} C_VEL
LIN {X 0,Y 181.386,Z 565.514,A -85,B 0,C 180,E1 -23338.968,E2 -23338.968} C_VEL
LIN {X 0,Y 185.16,Z 554.922,A -85,B 0,C 180,E1 -23341.46,E2 -23341.46} C_VEL
LIN {X 0,Y 188.882,Z 543.354,A -85,B 0,C 180,E1 -23343.606,E2 -23343.606} C_VEL
LIN {X 0,Y 192.393,Z 530.632,A -85,B 0,C 180,E1 -23345.444,E2 -23345.444} C_VEL
LIN {X 0,Y 195.367,Z 517.428,A -85,B 0,C 180,E1 -23346.892,E2 -23346.892} C_VEL
LIN {X 0,Y 197.799,Z 503.043,A -85,B 0,C 180,E1 -23348.042,E2 -23348.042} C_VEL
LIN {X 0,Y 199.374,Z 488.478,A -85,B 0,C 180,E1 -23348.814,E2 -23348.814} C_VEL
LIN {X 0,Y 203.381,Z 424.864,A -85,B 0,C 180,E1 -23350.834,E2 -23350.834} C_VEL
LIN {X 0,Y 200.439,Z 417.8,A -85,B 0,C 180,E1 -23351.992,E2 -23351.992} C_VEL
LIN {X 0,Y 194.494,Z 406.68,A -85,B 0,C 180,E1 -23354.35,E2 -23354.35} C_VEL
LIN {X 0,Y 187.47,Z 395.135,A -85,B 0,C 180,E1 -23357.394,E2 -23357.394} C_VEL
LIN {X 0,Y 181.868,Z 387.062,A -85,B 0,C 180,E1 -23360.077,E2 -23360.077} C_VEL
LIN {X 0,Y 179.013,Z 383.119,A -85,B 0,C 180,E1 -23361.567,E2 -23361.567} C_VEL
LIN {X 0,Y 176.065,Z 379.055,A -85,B 0,C 180,E1 -23363.218,E2 -23363.218} C_VEL
LIN {X 0,Y 173.482,Z 375.806,A -85,B 0,C 180,E1 -23364.75,E2 -23364.75} C_VEL
LIN {X 0,Y 172.49,Z 374.39,A -85,B 0,C 180,E1 -23365.382,E2 -23365.382} C_VEL
LIN {X 0,Y 169.951,Z 371.677,A -85,B 0,C 180,E1 -23367.011,E2 -23367.011} C_VEL
LIN {X 0,Y 168.776,Z 369.34,A -85,B 0,C 180,E1 -23367.902,E2 -23367.902} C_VEL
LIN {X 0,Y 166.204,Z 367.571,A -85,B 0,C 180,E1 -23369.682,E2 -23369.682} C_VEL
LIN {X 0,Y 164.681,Z 365.053,A -85,B 0,C 180,E1 -23370.957,E2 -23370.957} C_VEL
LIN {X 0,Y 164.327,Z 363.627,A -85,B 0,C 180,E1 -23371.413,E2 -23371.413} C_VEL
LIN {X 0,Y 164.387,Z 363.63,A -85,B 0,C 180,E1 -23374.688,E2 -23374.688} C_VEL
LIN {X 0,Y 164.418,Z 363.585,A -85,B 0,C 180,E1 -23380.117,E2 -23380.117} C_VEL
LIN {X 0,Y 164.48,Z 363.616,A -85,B 0,C 180,E1 -23385.144,E2 -23385.144} C_VEL
LIN {X 0,Y 164.766,Z 363.539,A -85,B 0,C 180,E1 -23390.176,E2 -23390.176} C_VEL
LIN {X 0,Y 164.824,Z 363.568,A -85,B 0,C 180,E1 -23392.65,E2 -23392.65} C_VEL
LIN {X 0,Y 165.04,Z 363.546,A -85,B 0,C 180,E1 -23397.559,E2 -23397.559} C_VEL
LIN {X 0,Y 165.277,Z 363.514,A -85,B 0,C 180,E1 -23399.999,E2 -23399.999} C_VEL
LIN {X 0,Y 164.823,Z 363.578,A -85,B 0,C 180,E1 -23407.349,E2 -23407.349} C_VEL
LIN {X 0,Y 164.704,Z 363.587,A -85,B 0,C 180,E1 -23411.059,E2 -23411.059} C_VEL
LIN {X 0,Y 164.485,Z 363.616,A -85,B 0,C 180,E1 -23417.402,E2 -23417.402} C_VEL
LIN {X 0,Y 164.474,Z 363.623,A -85,B 0,C 180,E1 -23419.988,E2 -23419.988} C_VEL
LIN {X 0,Y 164.387,Z 363.631,A -85,B 0,C 180,E1 -23423.294,E2 -23423.294} C_VEL
LIN {X 0,Y 165.226,Z 366.181,A -85,B 0,C 180,E1 -23424.167,E2 -23424.167} C_VEL
LIN {X 0,Y 167.153,Z 368.396,A -85,B 0,C 180,E1 -23425.647,E2 -23425.647} C_VEL
LIN {X 0,Y 168.922,Z 369.671,A -85,B 0,C 180,E1 -23426.854,E2 -23426.854} C_VEL
LIN {X 0,Y 170.642,Z 372.633,A -85,B 0,C 180,E1 -23428.102,E2 -23428.102} C_VEL
LIN {X 0,Y 173.11,Z 375.076,A -85,B 0,C 180,E1 -23429.639,E2 -23429.639} C_VEL
LIN {X 0,Y 175.703,Z 378.69,A -85,B 0,C 180,E1 -23431.219,E2 -23431.219} C_VEL
LIN {X 0,Y 177.081,Z 380.38,A -85,B 0,C 180,E1 -23431.998,E2 -23431.998} C_VEL
LIN {X 0,Y 180.832,Z 385.519,A -85,B 0,C 180,E1 -23434.024,E2 -23434.024} C_VEL
LIN {X 0,Y 183.422,Z 389.256,A -85,B 0,C 180,E1 -23435.335,E2 -23435.335} C_VEL
LIN {X 0,Y 188.591,Z 398.484,A -85,B 0,C 180,E1 -23437.845,E2 -23437.845} C_VEL
LIN {X 0,Y 194.034,Z 409.312,A -85,B 0,C 180,E1 -23440.282,E2 -23440.282} C_VEL
LIN {X 0,Y 199.406,Z 421.859,A -85,B 0,C 180,E1 -23442.553,E2 -23442.553} C_VEL
LIN {X 0,Y 203.086,Z 431.836,A -85,B 0,C 180,E1 -23444.058,E2 -23444.058} C_VEL
LIN {X 0,Y 198.893,Z 498.354,A -85,B 0,C 180,E1 -23446.183,E2 -23446.183} C_VEL
LIN {X 0,Y 197.09,Z 512.421,A -85,B 0,C 180,E1 -23446.914,E2 -23446.914} C_VEL
LIN {X 0,Y 195.628,Z 520.979,A -85,B 0,C 180,E1 -23447.548,E2 -23447.548} C_VEL
LIN {X 0,Y 194.373,Z 524.709,A -85,B 0,C 180,E1 -23447.727,E2 -23447.727} C_VEL
LIN {X 0,Y 187.288,Z 536.233,A -85,B 0,C 180,E1 -23447.833,E2 -23447.833} C_VEL
LIN {X 0,Y 185.794,Z 539.768,A -85,B 0,C 180,E1 -23448.14,E2 -23448.14} C_VEL
LIN {X 0,Y 181.86,Z 552.677,A -85,B 0,C 180,E1 -23450.023,E2 -23450.023} C_VEL
LIN {X 0,Y 178.196,Z 563.442,A -85,B 0,C 180,E1 -23452.072,E2 -23452.072} C_VEL
LIN {X 0,Y 173.755,Z 574.852,A -85,B 0,C 180,E1 -23454.803,E2 -23454.803} C_VEL
LIN {X 0,Y 169.235,Z 585.381,A -85,B 0,C 180,E1 -23458.029,E2 -23458.029} C_VEL
LIN {X 0,Y 165.319,Z 594.067,A -85,B 0,C 180,E1 -23461.428,E2 -23461.428} C_VEL
LIN {X 0,Y 161.552,Z 602.384,A -85,B 0,C 180,E1 -23465.59,E2 -23465.59} C_VEL
LIN {X 0,Y 159.121,Z 608.203,A -85,B 0,C 180,E1 -23469.308,E2 -23469.308} C_VEL
LIN {X 0,Y 157.133,Z 612.959,A -85,B 0,C 180,E1 -23473.099,E2 -23473.099} C_VEL
LIN {X 0,Y 155.454,Z 617.884,A -85,B 0,C 180,E1 -23478.262,E2 -23478.262} C_VEL
LIN {X 0,Y 154.859,Z 620.564,A -85,B 0,C 180,E1 -23482.175,E2 -23482.175} C_VEL
LIN {X 0,Y 154.696,Z 622.896,A -85,B 0,C 180,E1 -23487.396,E2 -23487.396} C_VEL
LIN {X 0,Y 154.808,Z 623.547,A -85,B 0,C 180,E1 -23490,E2 -23490} C_VEL
LIN {X 0,Y 154.688,Z 623.818,A -85,B 0,C 180,E1 -23495.214,E2 -23495.214} C_VEL
LIN {X 0,Y 155.268,Z 622.762,A -85,B 0,C 180,E1 -23500.431,E2 -23500.431} C_VEL
LIN {X 0,Y 156.728,Z 620.369,A -85,B 0,C 180,E1 -23505.608,E2 -23505.608} C_VEL
LIN {X 0,Y 159.44,Z 616.589,A -85,B 0,C 180,E1 -23510.649,E2 -23510.649} C_VEL
LIN {X 0,Y 163.131,Z 611.302,A -85,B 0,C 180,E1 -23515.52,E2 -23515.52} C_VEL
LIN {X 0,Y 166.708,Z 606.205,A -85,B 0,C 180,E1 -23519,E2 -23519} C_VEL
LIN {X 0,Y 171.701,Z 598.953,A -85,B 0,C 180,E1 -23522.844,E2 -23522.844} C_VEL
LIN {X 0,Y 177.387,Z 590.003,A -85,B 0,C 180,E1 -23526.463,E2 -23526.463} C_VEL
LIN {X 0,Y 182.849,Z 580.627,A -85,B 0,C 180,E1 -23529.361,E2 -23529.361} C_VEL
LIN {X 0,Y 188.632,Z 569.2,A -85,B 0,C 180,E1 -23532.117,E2 -23532.117} C_VEL
LIN {X 0,Y 193.846,Z 557.573,A -85,B 0,C 180,E1 -23534.261,E2 -23534.261} C_VEL
LIN {X 0,Y 198.256,Z 546.242,A -85,B 0,C 180,E1 -23535.877,E2 -23535.877} C_VEL
LIN {X 0,Y 202.298,Z 533.991,A -85,B 0,C 180,E1 -23537.215,E2 -23537.215} C_VEL
LIN {X 0,Y 205.828,Z 520.467,A -85,B 0,C 180,E1 -23538.325,E2 -23538.325} C_VEL
LIN {X 0,Y 208.478,Z 506.58,A -85,B 0,C 180,E1 -23539.141,E2 -23539.141} C_VEL
LIN {X 0,Y 210.265,Z 491.871,A -85,B 0,C 180,E1 -23539.693,E2 -23539.693} C_VEL
LIN {X 0,Y 213.522,Z 447.209,A -85,B 0,C 180,E1 -23540.988,E2 -23540.988} C_VEL
LIN {X 0,Y 208.824,Z 435.708,A -85,B 0,C 180,E1 -23543.422,E2 -23543.422} C_VEL
LIN {X 0,Y 203.831,Z 425.043,A -85,B 0,C 180,E1 -23546.222,E2 -23546.222} C_VEL
LIN {X 0,Y 199.064,Z 415.962,A -85,B 0,C 180,E1 -23549.19,E2 -23549.19} C_VEL
LIN {X 0,Y 195.999,Z 410.478,A -85,B 0,C 180,E1 -23551.314,E2 -23551.314} C_VEL
LIN {X 0,Y 192.904,Z 405.437,A -85,B 0,C 180,E1 -23553.667,E2 -23553.667} C_VEL
LIN {X 0,Y 191.438,Z 403.317,A -85,B 0,C 180,E1 -23554.864,E2 -23554.864} C_VEL
LIN {X 0,Y 188.237,Z 398.962,A -85,B 0,C 180,E1 -23557.76,E2 -23557.76} C_VEL
LIN {X 0,Y 185.528,Z 395.566,A -85,B 0,C 180,E1 -23560.63,E2 -23560.63} C_VEL
LIN {X 0,Y 184.744,Z 394.155,A -85,B 0,C 180,E1 -23561.628,E2 -23561.628} C_VEL
LIN {X 0,Y 182.104,Z 391.547,A -85,B 0,C 180,E1 -23565.258,E2 -23565.258} C_VEL
LIN {X 0,Y 180.775,Z 388.8,A -85,B 0,C 180,E1 -23567.939,E2 -23567.939} C_VEL
LIN {X 0,Y 178.459,Z 387.296,A -85,B 0,C 180,E1 -23575.483,E2 -23575.483} C_VEL
LIN {X 0,Y 178.519,Z 386.849,A -85,B 0,C 180,E1 -23580.001,E2 -23580.001} C_VEL
LIN {X 0,Y 181.008,Z 388.959,A -85,B 0,C 180,E1 -23587.951,E2 -23587.951} C_VEL
LIN {X 0,Y 182.479,Z 392.079,A -85,B 0,C 180,E1 -23590.79,E2 -23590.79} C_VEL
LIN {X 0,Y 185.018,Z 394.561,A -85,B 0,C 180,E1 -23594.155,E2 -23594.155} C_VEL
LIN {X 0,Y 187.235,Z 398.015,A -85,B 0,C 180,E1 -23596.71,E2 -23596.71} C_VEL
LIN {X 0,Y 188.757,Z 399.633,A -85,B 0,C 180,E1 -23598.178,E2 -23598.178} C_VEL
LIN {X 0,Y 191.627,Z 403.504,A -85,B 0,C 180,E1 -23600.724,E2 -23600.724} C_VEL
LIN {X 0,Y 195.582,Z 409.115,A -85,B 0,C 180,E1 -23603.766,E2 -23603.766} C_VEL
LIN {X 0,Y 200.409,Z 416.234,A -85,B 0,C 180,E1 -23606.963,E2 -23606.963} C_VEL
LIN {X 0,Y 205.462,Z 424.5,A -85,B 0,C 180,E1 -23609.912,E2 -23609.912} C_VEL
LIN {X 0,Y 210.758,Z 433.918,A -85,B 0,C 180,E1 -23612.671,E2 -23612.671} C_VEL
LIN {X 0,Y 214.007,Z 441.089,A -85,B 0,C 180,E1 -23614.287,E2 -23614.287} C_VEL
LIN {X 0,Y 210.204,Z 490.836,A -85,B 0,C 180,E1 -23615.742,E2 -23615.742} C_VEL
LIN {X 0,Y 208.092,Z 505.421,A -85,B 0,C 180,E1 -23616.463,E2 -23616.463} C_VEL
LIN {X 0,Y 205.217,Z 518.898,A -85,B 0,C 180,E1 -23617.429,E2 -23617.429} C_VEL
LIN {X 0,Y 201.454,Z 532.048,A -85,B 0,C 180,E1 -23618.685,E2 -23618.685} C_VEL
LIN {X 0,Y 197.898,Z 542.536,A -85,B 0,C 180,E1 -23620.009,E2 -23620.009} C_VEL
LIN {X 0,Y 192.86,Z 555.112,A -85,B 0,C 180,E1 -23622.056,E2 -23622.056} C_VEL
LIN {X 0,Y 188.163,Z 564.895,A -85,B 0,C 180,E1 -23624.028,E2 -23624.028} C_VEL
LIN {X 0,Y 183.439,Z 574.066,A -85,B 0,C 180,E1 -23626.399,E2 -23626.399} C_VEL
LIN {X 0,Y 178.236,Z 583.235,A -85,B 0,C 180,E1 -23629.412,E2 -23629.412} C_VEL
LIN {X 0,Y 173.312,Z 590.851,A -85,B 0,C 180,E1 -23632.535,E2 -23632.535} C_VEL
LIN {X 0,Y 168.953,Z 597.182,A -85,B 0,C 180,E1 -23635.835,E2 -23635.835} C_VEL
LIN {X 0,Y 165.217,Z 602.358,A -85,B 0,C 180,E1 -23639.306,E2 -23639.306} C_VEL
LIN {X 0,Y 161.114,Z 607.796,A -85,B 0,C 180,E1 -23644.137,E2 -23644.137} C_VEL
LIN {X 0,Y 158.058,Z 611.631,A -85,B 0,C 180,E1 -23649.162,E2 -23649.162} C_VEL
LIN {X 0,Y 155.973,Z 614.034,A -85,B 0,C 180,E1 -23654.314,E2 -23654.314} C_VEL
LIN {X 0,Y 154.908,Z 615.085,A -85,B 0,C 180,E1 -23659.544,E2 -23659.544} C_VEL
LIN {X 0,Y 154.682,Z 614.814,A -85,B 0,C 180,E1 -23664.786,E2 -23664.786} C_VEL
LIN {X 0,Y 154.891,Z 613.235,A -85,B 0,C 180,E1 -23670,E2 -23670} C_VEL
LIN {X 0,Y 155.715,Z 610.317,A -85,B 0,C 180,E1 -23675.179,E2 -23675.179} C_VEL
LIN {X 0,Y 157.442,Z 605.974,A -85,B 0,C 180,E1 -23680.286,E2 -23680.286} C_VEL
LIN {X 0,Y 160.121,Z 600.065,A -85,B 0,C 180,E1 -23685.269,E2 -23685.269} C_VEL
LIN {X 0,Y 163.034,Z 593.423,A -85,B 0,C 180,E1 -23689.517,E2 -23689.517} C_VEL
LIN {X 0,Y 166.261,Z 586.457,A -85,B 0,C 180,E1 -23693.017,E2 -23693.017} C_VEL
LIN {X 0,Y 170.265,Z 578.079,A -85,B 0,C 180,E1 -23696.342,E2 -23696.342} C_VEL
LIN {X 0,Y 174.586,Z 567.997,A -85,B 0,C 180,E1 -23699.546,E2 -23699.546} C_VEL
LIN {X 0,Y 178.415,Z 557.868,A -85,B 0,C 180,E1 -23702.126,E2 -23702.126} C_VEL
LIN {X 0,Y 181.304,Z 549.465,A -85,B 0,C 180,E1 -23703.864,E2 -23703.864} C_VEL
LIN {X 0,Y 184.877,Z 538.136,A -85,B 0,C 180,E1 -23705.766,E2 -23705.766} C_VEL
LIN {X 0,Y 188.084,Z 525.889,A -85,B 0,C 180,E1 -23707.388,E2 -23707.388} C_VEL
LIN {X 0,Y 190.993,Z 512.321,A -85,B 0,C 180,E1 -23708.723,E2 -23708.723} C_VEL
LIN {X 0,Y 193.114,Z 498.265,A -85,B 0,C 180,E1 -23709.729,E2 -23709.729} C_VEL
LIN {X 0,Y 194.458,Z 484.924,A -85,B 0,C 180,E1 -23710.328,E2 -23710.328} C_VEL
LIN {X 0,Y 198.143,Z 426.958,A -85,B 0,C 180,E1 -23712.193,E2 -23712.193} C_VEL
LIN {X 0,Y 195.267,Z 420.372,A -85,B 0,C 180,E1 -23713.387,E2 -23713.387} C_VEL
LIN {X 0,Y 189.617,Z 409.814,A -85,B 0,C 180,E1 -23715.79,E2 -23715.79} C_VEL
LIN {X 0,Y 183.43,Z 399.632,A -85,B 0,C 180,E1 -23718.656,E2 -23718.656} C_VEL
LIN {X 0,Y 178.173,Z 391.847,A -85,B 0,C 180,E1 -23721.353,E2 -23721.353} C_VEL
LIN {X 0,Y 175.291,Z 387.901,A -85,B 0,C 180,E1 -23722.958,E2 -23722.958} C_VEL
LIN {X 0,Y 173.337,Z 385.015,A -85,B 0,C 180,E1 -23724.134,E2 -23724.134} C_VEL
LIN {X 0,Y 170.586,Z 381.32,A -85,B 0,C 180,E1 -23725.873,E2 -23725.873} C_VEL
LIN {X 0,Y 167.237,Z 377.312,A -85,B 0,C 180,E1 -23728.156,E2 -23728.156} C_VEL
LIN {X 0,Y 166.195,Z 375.685,A -85,B 0,C 180,E1 -23728.954,E2 -23728.954} C_VEL
LIN {X 0,Y 163.513,Z 373.192,A -85,B 0,C 180,E1 -23730.994,E2 -23730.994} C_VEL
LIN {X 0,Y 161.843,Z 370.273,A -85,B 0,C 180,E1 -23732.522,E2 -23732.522} C_VEL
LIN {X 0,Y 159.075,Z 368.365,A -85,B 0,C 180,E1 -23735.008,E2 -23735.008} C_VEL
LIN {X 0,Y 157.649,Z 366.038,A -85,B 0,C 180,E1 -23736.606,E2 -23736.606} C_VEL
LIN {X 0,Y 157.31,Z 364.489,A -85,B 0,C 180,E1 -23737.161,E2 -23737.161} C_VEL
LIN {X 0,Y 157.359,Z 364.475,A -85,B 0,C 180,E1 -23741.781,E2 -23741.781} C_VEL
LIN {X 0,Y 157.498,Z 364.451,A -85,B 0,C 180,E1 -23747.107,E2 -23747.107} C_VEL
LIN {X 0,Y 157.689,Z 364.417,A -85,B 0,C 180,E1 -23749.73,E2 -23749.73} C_VEL
LIN {X 0,Y 157.762,Z 364.439,A -85,B 0,C 180,E1 -23752.319,E2 -23752.319} C_VEL
LIN {X 0,Y 158.239,Z 364.391,A -85,B 0,C 180,E1 -23759.999,E2 -23759.999} C_VEL
LIN {X 0,Y 157.762,Z 364.459,A -85,B 0,C 180,E1 -23767.68,E2 -23767.68} C_VEL
LIN {X 0,Y 157.638,Z 364.468,A -85,B 0,C 180,E1 -23771.236,E2 -23771.236} C_VEL
LIN {X 0,Y 157.427,Z 364.501,A -85,B 0,C 180,E1 -23777.621,E2 -23777.621} C_VEL
LIN {X 0,Y 158.122,Z 366.804,A -85,B 0,C 180,E1 -23778.579,E2 -23778.579} C_VEL
LIN {X 0,Y 160.051,Z 369.22,A -85,B 0,C 180,E1 -23780.565,E2 -23780.565} C_VEL
LIN {X 0,Y 162.148,Z 370.503,A -85,B 0,C 180,E1 -23782.371,E2 -23782.371} C_VEL
LIN {X 0,Y 163.898,Z 373.625,A -85,B 0,C 180,E1 -23783.955,E2 -23783.955} C_VEL
LIN {X 0,Y 166.633,Z 376.201,A -85,B 0,C 180,E1 -23786.009,E2 -23786.009} C_VEL
LIN {X 0,Y 168.839,Z 379.485,A -85,B 0,C 180,E1 -23787.628,E2 -23787.628} C_VEL
LIN {X 0,Y 170.608,Z 381.328,A -85,B 0,C 180,E1 -23788.78,E2 -23788.78} C_VEL
LIN {X 0,Y 173.423,Z 385.087,A -85,B 0,C 180,E1 -23790.554,E2 -23790.554} C_VEL
LIN {X 0,Y 178.155,Z 391.731,A -85,B 0,C 180,E1 -23793.269,E2 -23793.269} C_VEL
LIN {X 0,Y 180.271,Z 394.958,A -85,B 0,C 180,E1 -23794.4,E2 -23794.4} C_VEL
LIN {X 0,Y 184.719,Z 403.088,A -85,B 0,C 180,E1 -23796.69,E2 -23796.69} C_VEL
LIN {X 0,Y 190.401,Z 414.772,A -85,B 0,C 180,E1 -23799.391,E2 -23799.391} C_VEL
LIN {X 0,Y 196.003,Z 428.607,A -85,B 0,C 180,E1 -23801.899,E2 -23801.899} C_VEL
LIN {X 0,Y 197.86,Z 433.872,A -85,B 0,C 180,E1 -23802.71,E2 -23802.71} C_VEL
LIN {X 0,Y 193.571,Z 498.699,A -85,B 0,C 180,E1 -23804.813,E2 -23804.813} C_VEL
LIN {X 0,Y 191.661,Z 512.851,A -85,B 0,C 180,E1 -23805.572,E2 -23805.572} C_VEL
LIN {X 0,Y 189.018,Z 526.904,A -85,B 0,C 180,E1 -23806.722,E2 -23806.722} C_VEL
LIN {X 0,Y 185.794,Z 539.768,A -85,B 0,C 180,E1 -23808.14,E2 -23808.14} C_VEL
LIN {X 0,Y 183.749,Z 545.042,A -85,B 0,C 180,E1 -23808.71,E2 -23808.71} C_VEL
LIN {X 0,Y 178.859,Z 553.341,A -85,B 0,C 180,E1 -23809.438,E2 -23809.438} C_VEL
LIN {X 0,Y 173.783,Z 561.306,A -85,B 0,C 180,E1 -23810.385,E2 -23810.385} C_VEL
LIN {X 0,Y 171.484,Z 565.962,A -85,B 0,C 180,E1 -23811.303,E2 -23811.303} C_VEL
LIN {X 0,Y 167.17,Z 576.286,A -85,B 0,C 180,E1 -23813.944,E2 -23813.944} C_VEL
LIN {X 0,Y 162.471,Z 586.481,A -85,B 0,C 180,E1 -23817.268,E2 -23817.268} C_VEL
LIN {X 0,Y 158.435,Z 594.947,A -85,B 0,C 180,E1 -23820.794,E2 -23820.794} C_VEL
LIN {X 0,Y 154.566,Z 603.034,A -85,B 0,C 180,E1 -23825.128,E2 -23825.128} C_VEL
LIN {X 0,Y 151.665,Z 609.55,A -85,B 0,C 180,E1 -23829.663,E2 -23829.663} C_VEL
LIN {X 0,Y 149.198,Z 615.313,A -85,B 0,C 180,E1 -23834.985,E2 -23834.985} C_VEL
LIN {X 0,Y 148.208,Z 618.594,A -85,B 0,C 180,E1 -23839.066,E2 -23839.066} C_VEL
LIN {X 0,Y 147.624,Z 621.657,A -85,B 0,C 180,E1 -23844.536,E2 -23844.536} C_VEL
LIN {X 0,Y 147.715,Z 623.326,A -85,B 0,C 180,E1 -23850,E2 -23850} C_VEL
LIN {X 0,Y 147.607,Z 623.642,A -85,B 0,C 180,E1 -23852.729,E2 -23852.729} C_VEL
LIN {X 0,Y 147.807,Z 623.272,A -85,B 0,C 180,E1 -23858.201,E2 -23858.201} C_VEL
LIN {X 0,Y 148.93,Z 621.578,A -85,B 0,C 180,E1 -23863.648,E2 -23863.648} C_VEL
LIN {X 0,Y 151.213,Z 618.529,A -85,B 0,C 180,E1 -23868.987,E2 -23868.987} C_VEL
LIN {X 0,Y 154.6,Z 614.042,A -85,B 0,C 180,E1 -23874.151,E2 -23874.151} C_VEL
LIN {X 0,Y 157.911,Z 609.616,A -85,B 0,C 180,E1 -23877.86,E2 -23877.86} C_VEL
LIN {X 0,Y 162.639,Z 603.238,A -85,B 0,C 180,E1 -23881.962,E2 -23881.962} C_VEL
LIN {X 0,Y 168.175,Z 595.328,A -85,B 0,C 180,E1 -23885.807,E2 -23885.807} C_VEL
LIN {X 0,Y 173.594,Z 587.076,A -85,B 0,C 180,E1 -23888.868,E2 -23888.868} C_VEL
LIN {X 0,Y 179.371,Z 577.156,A -85,B 0,C 180,E1 -23891.766,E2 -23891.766} C_VEL
LIN {X 0,Y 185.016,Z 566.143,A -85,B 0,C 180,E1 -23894.266,E2 -23894.266} C_VEL
LIN {X 0,Y 190.535,Z 553.87,A -85,B 0,C 180,E1 -23896.376,E2 -23896.376} C_VEL
LIN {X 0,Y 195.168,Z 541.722,A -85,B 0,C 180,E1 -23897.963,E2 -23897.963} C_VEL
LIN {X 0,Y 199.388,Z 528.241,A -85,B 0,C 180,E1 -23899.274,E2 -23899.274} C_VEL
LIN {X 0,Y 202.728,Z 514.065,A -85,B 0,C 180,E1 -23900.292,E2 -23900.292} C_VEL
LIN {X 0,Y 205.087,Z 499.904,A -85,B 0,C 180,E1 -23900.971,E2 -23900.971} C_VEL
LIN {X 0,Y 207.267,Z 475.105,A -85,B 0,C 180,E1 -23901.72,E2 -23901.72} C_VEL
LIN {X 0,Y 209.121,Z 449.833,A -85,B 0,C 180,E1 -23902.474,E2 -23902.474} C_VEL
LIN {X 0,Y 205.038,Z 439.579,A -85,B 0,C 180,E1 -23904.753,E2 -23904.753} C_VEL
LIN {X 0,Y 200.504,Z 429.623,A -85,B 0,C 180,E1 -23907.482,E2 -23907.482} C_VEL
LIN {X 0,Y 196.127,Z 420.983,A -85,B 0,C 180,E1 -23910.409,E2 -23910.409} C_VEL
LIN {X 0,Y 192.365,Z 414.038,A -85,B 0,C 180,E1 -23913.258,E2 -23913.258} C_VEL
LIN {X 0,Y 189.566,Z 409.745,A -85,B 0,C 180,E1 -23915.601,E2 -23915.601} C_VEL
LIN {X 0,Y 186.441,Z 405.385,A -85,B 0,C 180,E1 -23918.582,E2 -23918.582} C_VEL
LIN {X 0,Y 183.87,Z 401.869,A -85,B 0,C 180,E1 -23921.507,E2 -23921.507} C_VEL
LIN {X 0,Y 183.18,Z 400.821,A -85,B 0,C 180,E1 -23922.415,E2 -23922.415} C_VEL
LIN {X 0,Y 180.682,Z 398.006,A -85,B 0,C 180,E1 -23926.164,E2 -23926.164} C_VEL
LIN {X 0,Y 179.692,Z 395.762,A -85,B 0,C 180,E1 -23928.344,E2 -23928.344} C_VEL
LIN {X 0,Y 177.496,Z 394.075,A -85,B 0,C 180,E1 -23937.164,E2 -23937.164} C_VEL
LIN {X 0,Y 177.711,Z 394.063,A -85,B 0,C 180,E1 -23940.567,E2 -23940.567} C_VEL
LIN {X 0,Y 179.862,Z 395.857,A -85,B 0,C 180,E1 -23947.438,E2 -23947.438} C_VEL
LIN {X 0,Y 181.504,Z 399.227,A -85,B 0,C 180,E1 -23950.69,E2 -23950.69} C_VEL
LIN {X 0,Y 183.599,Z 401.308,A -85,B 0,C 180,E1 -23953.56,E2 -23953.56} C_VEL
LIN {X 0,Y 185.953,Z 404.935,A -85,B 0,C 180,E1 -23956.367,E2 -23956.367} C_VEL
LIN {X 0,Y 187.303,Z 406.586,A -85,B 0,C 180,E1 -23957.731,E2 -23957.731} C_VEL
LIN {X 0,Y 190.553,Z 411.163,A -85,B 0,C 180,E1 -23960.688,E2 -23960.688} C_VEL
LIN {X 0,Y 194.006,Z 416.208,A -85,B 0,C 180,E1 -23963.4,E2 -23963.4} C_VEL
LIN {X 0,Y 198.649,Z 423.431,A -85,B 0,C 180,E1 -23966.579,E2 -23966.579} C_VEL
LIN {X 0,Y 203.381,Z 431.405,A -85,B 0,C 180,E1 -23969.43,E2 -23969.43} C_VEL
LIN {X 0,Y 208.324,Z 440.791,A -85,B 0,C 180,E1 -23972.118,E2 -23972.118} C_VEL
LIN {X 0,Y 209.584,Z 443.764,A -85,B 0,C 180,E1 -23972.789,E2 -23972.789} C_VEL
LIN {X 0,Y 205.788,Z 491.723,A -85,B 0,C 180,E1 -23974.223,E2 -23974.223} C_VEL
LIN {X 0,Y 203.623,Z 506.023,A -85,B 0,C 180,E1 -23974.942,E2 -23974.942} C_VEL
LIN {X 0,Y 200.355,Z 520.533,A -85,B 0,C 180,E1 -23976.003,E2 -23976.003} C_VEL
LIN {X 0,Y 196.475,Z 533.369,A -85,B 0,C 180,E1 -23977.26,E2 -23977.26} C_VEL
LIN {X 0,Y 192.456,Z 544.542,A -85,B 0,C 180,E1 -23978.724,E2 -23978.724} C_VEL
LIN {X 0,Y 187.588,Z 556.054,A -85,B 0,C 180,E1 -23980.653,E2 -23980.653} C_VEL
LIN {X 0,Y 182.227,Z 566.693,A -85,B 0,C 180,E1 -23982.88,E2 -23982.88} C_VEL
LIN {X 0,Y 176.373,Z 577.32,A -85,B 0,C 180,E1 -23985.829,E2 -23985.829} C_VEL
LIN {X 0,Y 171.028,Z 585.9,A -85,B 0,C 180,E1 -23988.891,E2 -23988.891} C_VEL
LIN {X 0,Y 165.284,Z 594.179,A -85,B 0,C 180,E1 -23992.705,E2 -23992.705} C_VEL
LIN {X 0,Y 160.129,Z 600.998,A -85,B 0,C 180,E1 -23996.914,E2 -23996.914} C_VEL
LIN {X 0,Y 155.625,Z 606.649,A -85,B 0,C 180,E1 -24001.694,E2 -24001.694} C_VEL
LIN {X 0,Y 152.882,Z 610.018,A -85,B 0,C 180,E1 -24005.56,E2 -24005.56} C_VEL
LIN {X 0,Y 150.059,Z 613.156,A -85,B 0,C 180,E1 -24010.862,E2 -24010.862} C_VEL
LIN {X 0,Y 148.301,Z 614.908,A -85,B 0,C 180,E1 -24016.293,E2 -24016.293} C_VEL
LIN {X 0,Y 147.666,Z 615.323,A -85,B 0,C 180,E1 -24021.791,E2 -24021.791} C_VEL
LIN {X 0,Y 147.645,Z 614.427,A -85,B 0,C 180,E1 -24027.272,E2 -24027.272} C_VEL
LIN {X 0,Y 148.124,Z 612.216,A -85,B 0,C 180,E1 -24032.719,E2 -24032.719} C_VEL
LIN {X 0,Y 149.418,Z 608.632,A -85,B 0,C 180,E1 -24038.112,E2 -24038.112} C_VEL
LIN {X 0,Y 151.134,Z 604.972,A -85,B 0,C 180,E1 -24042.079,E2 -24042.079} C_VEL
LIN {X 0,Y 153.299,Z 600.422,A -85,B 0,C 180,E1 -24045.966,E2 -24045.966} C_VEL
LIN {X 0,Y 156.385,Z 593.824,A -85,B 0,C 180,E1 -24050.383,E2 -24050.383} C_VEL
LIN {X 0,Y 160.436,Z 585.601,A -85,B 0,C 180,E1 -24054.592,E2 -24054.592} C_VEL
LIN {X 0,Y 164.636,Z 577.02,A -85,B 0,C 180,E1 -24058.006,E2 -24058.006} C_VEL
LIN {X 0,Y 169.174,Z 566.638,A -85,B 0,C 180,E1 -24061.285,E2 -24061.285} C_VEL
LIN {X 0,Y 173.269,Z 556.195,A -85,B 0,C 180,E1 -24063.898,E2 -24063.898} C_VEL
LIN {X 0,Y 177.293,Z 544.814,A -85,B 0,C 180,E1 -24066.133,E2 -24066.133} C_VEL
LIN {X 0,Y 181.063,Z 532.346,A -85,B 0,C 180,E1 -24068.039,E2 -24068.039} C_VEL
LIN {X 0,Y 184.551,Z 518.379,A -85,B 0,C 180,E1 -24069.633,E2 -24069.633} C_VEL
LIN {X 0,Y 187.166,Z 504.228,A -85,B 0,C 180,E1 -24070.813,E2 -24070.813} C_VEL
LIN {X 0,Y 188.865,Z 490.309,A -85,B 0,C 180,E1 -24071.606,E2 -24071.606} C_VEL
LIN {X 0,Y 193.077,Z 429.236,A -85,B 0,C 180,E1 -24073.599,E2 -24073.599} C_VEL
LIN {X 0,Y 188.046,Z 418.741,A -85,B 0,C 180,E1 -24075.827,E2 -24075.827} C_VEL
LIN {X 0,Y 181.842,Z 407.884,A -85,B 0,C 180,E1 -24078.771,E2 -24078.771} C_VEL
LIN {X 0,Y 176.464,Z 399.327,A -85,B 0,C 180,E1 -24081.612,E2 -24081.612} C_VEL
LIN {X 0,Y 170.566,Z 390.916,A -85,B 0,C 180,E1 -24085.13,E2 -24085.13} C_VEL
LIN {X 0,Y 167.278,Z 386.505,A -85,B 0,C 180,E1 -24087.345,E2 -24087.345} C_VEL
LIN {X 0,Y 164.535,Z 382.83,A -85,B 0,C 180,E1 -24089.386,E2 -24089.386} C_VEL
LIN {X 0,Y 163.511,Z 381.725,A -85,B 0,C 180,E1 -24090.177,E2 -24090.177} C_VEL
LIN {X 0,Y 161.015,Z 378.835,A -85,B 0,C 180,E1 -24092.269,E2 -24092.269} C_VEL
LIN {X 0,Y 159.937,Z 376.952,A -85,B 0,C 180,E1 -24093.314,E2 -24093.314} C_VEL
LIN {X 0,Y 157.071,Z 374.583,A -85,B 0,C 180,E1 -24096.085,E2 -24096.085} C_VEL
LIN {X 0,Y 155.573,Z 371.755,A -85,B 0,C 180,E1 -24097.943,E2 -24097.943} C_VEL
LIN {X 0,Y 155.199,Z 371.255,A -85,B 0,C 180,E1 -24098.411,E2 -24098.411} C_VEL
LIN {X 0,Y 152.119,Z 369.287,A -85,B 0,C 180,E1 -24102.523,E2 -24102.523} C_VEL
LIN {X 0,Y 150.688,Z 366.775,A -85,B 0,C 180,E1 -24105.308,E2 -24105.308} C_VEL
LIN {X 0,Y 150.405,Z 365.344,A -85,B 0,C 180,E1 -24106.316,E2 -24106.316} C_VEL
LIN {X 0,Y 150.608,Z 365.297,A -85,B 0,C 180,E1 -24109.241,E2 -24109.241} C_VEL
LIN {X 0,Y 150.685,Z 365.312,A -85,B 0,C 180,E1 -24111.956,E2 -24111.956} C_VEL
LIN {X 0,Y 151.2,Z 365.267,A -85,B 0,C 180,E1 -24119.999,E2 -24119.999} C_VEL
LIN {X 0,Y 150.653,Z 365.339,A -85,B 0,C 180,E1 -24128.72,E2 -24128.72} C_VEL
LIN {X 0,Y 150.797,Z 366.17,A -85,B 0,C 180,E1 -24129.387,E2 -24129.387} C_VEL
LIN {X 0,Y 152.005,Z 368.871,A -85,B 0,C 180,E1 -24131.874,E2 -24131.874} C_VEL
LIN {X 0,Y 154.311,Z 370.86,A -85,B 0,C 180,E1 -24135.181,E2 -24135.181} C_VEL
LIN {X 0,Y 155.632,Z 371.538,A -85,B 0,C 180,E1 -24136.73,E2 -24136.73} C_VEL
LIN {X 0,Y 157.025,Z 374.376,A -85,B 0,C 180,E1 -24138.485,E2 -24138.485} C_VEL
LIN {X 0,Y 159.539,Z 376.711,A -85,B 0,C 180,E1 -24140.972,E2 -24140.972} C_VEL
LIN {X 0,Y 160.266,Z 377.369,A -85,B 0,C 180,E1 -24141.631,E2 -24141.631} C_VEL
LIN {X 0,Y 162.41,Z 380.656,A -85,B 0,C 180,E1 -24143.584,E2 -24143.584} C_VEL
LIN {X 0,Y 164.31,Z 382.466,A -85,B 0,C 180,E1 -24145.069,E2 -24145.069} C_VEL
LIN {X 0,Y 166.92,Z 386.136,A -85,B 0,C 180,E1 -24147.048,E2 -24147.048} C_VEL
LIN {X 0,Y 168.239,Z 387.681,A -85,B 0,C 180,E1 -24147.957,E2 -24147.957} C_VEL
LIN {X 0,Y 172.15,Z 393.158,A -85,B 0,C 180,E1 -24150.509,E2 -24150.509} C_VEL
LIN {X 0,Y 175.291,Z 397.615,A -85,B 0,C 180,E1 -24152.367,E2 -24152.367} C_VEL
LIN {X 0,Y 178.163,Z 402.304,A -85,B 0,C 180,E1 -24153.98,E2 -24153.98} C_VEL
LIN {X 0,Y 183.948,Z 413.901,A -85,B 0,C 180,E1 -24157.049,E2 -24157.049} C_VEL
LIN {X 0,Y 188.56,Z 424.61,A -85,B 0,C 180,E1 -24159.317,E2 -24159.317} C_VEL
LIN {X 0,Y 192.734,Z 435.908,A -85,B 0,C 180,E1 -24161.285,E2 -24161.285} C_VEL
LIN {X 0,Y 188.405,Z 498.741,A -85,B 0,C 180,E1 -24163.357,E2 -24163.357} C_VEL
LIN {X 0,Y 186.494,Z 512.519,A -85,B 0,C 180,E1 -24164.104,E2 -24164.104} C_VEL
LIN {X 0,Y 183.844,Z 525.955,A -85,B 0,C 180,E1 -24165.184,E2 -24165.184} C_VEL
LIN {X 0,Y 180.47,Z 539.218,A -85,B 0,C 180,E1 -24166.657,E2 -24166.657} C_VEL
LIN {X 0,Y 176.42,Z 552.004,A -85,B 0,C 180,E1 -24168.525,E2 -24168.525} C_VEL
LIN {X 0,Y 172.172,Z 563.993,A -85,B 0,C 180,E1 -24170.856,E2 -24170.856} C_VEL
LIN {X 0,Y 171.484,Z 565.962,A -85,B 0,C 180,E1 -24171.303,E2 -24171.303} C_VEL
LIN {X 0,Y 169.119,Z 570.59,A -85,B 0,C 180,E1 -24172.303,E2 -24172.303} C_VEL
LIN {X 0,Y 163.588,Z 577.704,A -85,B 0,C 180,E1 -24173.731,E2 -24173.731} C_VEL
LIN {X 0,Y 157.914,Z 584.385,A -85,B 0,C 180,E1 -24175.376,E2 -24175.376} C_VEL
LIN {X 0,Y 155.379,Z 588.222,A -85,B 0,C 180,E1 -24176.709,E2 -24176.709} C_VEL
LIN {X 0,Y 150.972,Z 597.032,A -85,B 0,C 180,E1 -24180.739,E2 -24180.739} C_VEL
LIN {X 0,Y 147.24,Z 604.387,A -85,B 0,C 180,E1 -24185.079,E2 -24185.079} C_VEL
LIN {X 0,Y 144.224,Z 610.848,A -85,B 0,C 180,E1 -24190.056,E2 -24190.056} C_VEL
LIN {X 0,Y 141.857,Z 616.226,A -85,B 0,C 180,E1 -24195.658,E2 -24195.658} C_VEL
LIN {X 0,Y 140.754,Z 620.042,A -85,B 0,C 180,E1 -24201.385,E2 -24201.385} C_VEL
LIN {X 0,Y 140.504,Z 622.428,A -85,B 0,C 180,E1 -24207.133,E2 -24207.133} C_VEL
LIN {X 0,Y 140.567,Z 623.21,A -85,B 0,C 180,E1 -24210.644,E2 -24210.644} C_VEL
LIN {X 0,Y 140.533,Z 623.427,A -85,B 0,C 180,E1 -24215.74,E2 -24215.74} C_VEL
LIN {X 0,Y 141.247,Z 622.421,A -85,B 0,C 180,E1 -24221.48,E2 -24221.48} C_VEL
LIN {X 0,Y 143.017,Z 620.082,A -85,B 0,C 180,E1 -24227.149,E2 -24227.149} C_VEL
LIN {X 0,Y 146.151,Z 616.356,A -85,B 0,C 180,E1 -24232.625,E2 -24232.625} C_VEL
LIN {X 0,Y 150.378,Z 611.137,A -85,B 0,C 180,E1 -24237.863,E2 -24237.863} C_VEL
LIN {X 0,Y 154.38,Z 606.095,A -85,B 0,C 180,E1 -24241.57,E2 -24241.57} C_VEL
LIN {X 0,Y 159.891,Z 598.912,A -85,B 0,C 180,E1 -24245.62,E2 -24245.62} C_VEL
LIN {X 0,Y 165.223,Z 591.407,A -85,B 0,C 180,E1 -24248.86,E2 -24248.86} C_VEL
LIN {X 0,Y 171.054,Z 582.482,A -85,B 0,C 180,E1 -24251.854,E2 -24251.854} C_VEL
LIN {X 0,Y 176.223,Z 573.496,A -85,B 0,C 180,E1 -24254.259,E2 -24254.259} C_VEL
LIN {X 0,Y 181.699,Z 562.869,A -85,B 0,C 180,E1 -24256.489,E2 -24256.489} C_VEL
LIN {X 0,Y 186.876,Z 551.296,A -85,B 0,C 180,E1 -24258.371,E2 -24258.371} C_VEL
LIN {X 0,Y 191.749,Z 538.576,A -85,B 0,C 180,E1 -24259.918,E2 -24259.918} C_VEL
LIN {X 0,Y 195.813,Z 525.401,A -85,B 0,C 180,E1 -24261.114,E2 -24261.114} C_VEL
LIN {X 0,Y 199.029,Z 511.491,A -85,B 0,C 180,E1 -24262.046,E2 -24262.046} C_VEL
LIN {X 0,Y 201.277,Z 497.139,A -85,B 0,C 180,E1 -24262.69,E2 -24262.69} C_VEL
LIN {X 0,Y 204.931,Z 452.601,A -85,B 0,C 180,E1 -24263.988,E2 -24263.988} C_VEL
LIN {X 0,Y 200.943,Z 442.43,A -85,B 0,C 180,E1 -24266.398,E2 -24266.398} C_VEL
LIN {X 0,Y 196.278,Z 432.036,A -85,B 0,C 180,E1 -24269.478,E2 -24269.478} C_VEL
LIN {X 0,Y 192.046,Z 423.607,A -85,B 0,C 180,E1 -24272.631,E2 -24272.631} C_VEL
LIN {X 0,Y 189.175,Z 418.383,A -85,B 0,C 180,E1 -24275.046,E2 -24275.046} C_VEL
LIN {X 0,Y 187.495,Z 415.884,A -85,B 0,C 180,E1 -24276.561,E2 -24276.561} C_VEL
LIN {X 0,Y 184.91,Z 412.055,A -85,B 0,C 180,E1 -24279.181,E2 -24279.181} C_VEL
LIN {X 0,Y 182.306,Z 408.279,A -85,B 0,C 180,E1 -24282.327,E2 -24282.327} C_VEL
LIN {X 0,Y 181.127,Z 406.957,A -85,B 0,C 180,E1 -24283.952,E2 -24283.952} C_VEL
LIN {X 0,Y 178.953,Z 403.657,A -85,B 0,C 180,E1 -24287.883,E2 -24287.883} C_VEL
LIN {X 0,Y 178.659,Z 402.776,A -85,B 0,C 180,E1 -24288.657,E2 -24288.657} C_VEL
LIN {X 0,Y 176.73,Z 401.4,A -85,B 0,C 180,E1 -24295.439,E2 -24295.439} C_VEL
LIN {X 0,Y 176.784,Z 400.954,A -85,B 0,C 180,E1 -24300.001,E2 -24300.001} C_VEL
LIN {X 0,Y 178.732,Z 402.742,A -85,B 0,C 180,E1 -24306.917,E2 -24306.917} C_VEL
LIN {X 0,Y 180.345,Z 406.113,A -85,B 0,C 180,E1 -24310.284,E2 -24310.284} C_VEL
LIN {X 0,Y 182.217,Z 408.091,A -85,B 0,C 180,E1 -24312.982,E2 -24312.982} C_VEL
LIN {X 0,Y 184.57,Z 411.734,A -85,B 0,C 180,E1 -24315.902,E2 -24315.902} C_VEL
LIN {X 0,Y 185.748,Z 413.333,A -85,B 0,C 180,E1 -24317.156,E2 -24317.156} C_VEL
LIN {X 0,Y 188.74,Z 417.681,A -85,B 0,C 180,E1 -24320.006,E2 -24320.006} C_VEL
LIN {X 0,Y 191.762,Z 422.205,A -85,B 0,C 180,E1 -24322.505,E2 -24322.505} C_VEL
LIN {X 0,Y 196.548,Z 429.959,A -85,B 0,C 180,E1 -24325.949,E2 -24325.949} C_VEL
LIN {X 0,Y 201.277,Z 438.408,A -85,B 0,C 180,E1 -24328.925,E2 -24328.925} C_VEL
LIN {X 0,Y 205.228,Z 446.292,A -85,B 0,C 180,E1 -24331.184,E2 -24331.184} C_VEL
LIN {X 0,Y 205.378,Z 446.646,A -85,B 0,C 180,E1 -24331.269,E2 -24331.269} C_VEL
LIN {X 0,Y 201.666,Z 491.623,A -85,B 0,C 180,E1 -24332.601,E2 -24332.601} C_VEL
LIN {X 0,Y 199.463,Z 505.862,A -85,B 0,C 180,E1 -24333.308,E2 -24333.308} C_VEL
LIN {X 0,Y 196.246,Z 519.897,A -85,B 0,C 180,E1 -24334.317,E2 -24334.317} C_VEL
LIN {X 0,Y 192.242,Z 532.916,A -85,B 0,C 180,E1 -24335.568,E2 -24335.568} C_VEL
LIN {X 0,Y 188.428,Z 543.262,A -85,B 0,C 180,E1 -24336.876,E2 -24336.876} C_VEL
LIN {X 0,Y 183.576,Z 554.641,A -85,B 0,C 180,E1 -24338.736,E2 -24338.736} C_VEL
LIN {X 0,Y 178.505,Z 564.572,A -85,B 0,C 180,E1 -24340.72,E2 -24340.72} C_VEL
LIN {X 0,Y 172.43,Z 575.321,A -85,B 0,C 180,E1 -24343.567,E2 -24343.567} C_VEL
LIN {X 0,Y 166.623,Z 584.491,A -85,B 0,C 180,E1 -24346.732,E2 -24346.732} C_VEL
LIN {X 0,Y 160.434,Z 593.074,A -85,B 0,C 180,E1 -24350.565,E2 -24350.565} C_VEL
LIN {X 0,Y 155.046,Z 599.952,A -85,B 0,C 180,E1 -24354.679,E2 -24354.679} C_VEL
LIN {X 0,Y 150.469,Z 605.423,A -85,B 0,C 180,E1 -24359.084,E2 -24359.084} C_VEL
LIN {X 0,Y 146.339,Z 610.13,A -85,B 0,C 180,E1 -24364.391,E2 -24364.391} C_VEL
LIN {X 0,Y 143.292,Z 613.307,A -85,B 0,C 180,E1 -24369.92,E2 -24369.92} C_VEL
LIN {X 0,Y 141.336,Z 615.089,A -85,B 0,C 180,E1 -24375.603,E2 -24375.603} C_VEL
LIN {X 0,Y 140.596,Z 615.533,A -85,B 0,C 180,E1 -24381.375,E2 -24381.375} C_VEL
LIN {X 0,Y 140.515,Z 615.262,A -85,B 0,C 180,E1 -24384.259,E2 -24384.259} C_VEL
LIN {X 0,Y 140.609,Z 614.276,A -85,B 0,C 180,E1 -24388.524,E2 -24388.524} C_VEL
LIN {X 0,Y 141.044,Z 612.485,A -85,B 0,C 180,E1 -24392.856,E2 -24392.856} C_VEL
LIN {X 0,Y 142.407,Z 608.932,A -85,B 0,C 180,E1 -24398.514,E2 -24398.514} C_VEL
LIN {X 0,Y 144.927,Z 603.893,A -85,B 0,C 180,E1 -24404.032,E2 -24404.032} C_VEL
LIN {X 0,Y 147.34,Z 599.02,A -85,B 0,C 180,E1 -24408.062,E2 -24408.062} C_VEL
LIN {X 0,Y 150.868,Z 592.029,A -85,B 0,C 180,E1 -24412.601,E2 -24412.601} C_VEL
LIN {X 0,Y 154.749,Z 584.707,A -85,B 0,C 180,E1 -24416.283,E2 -24416.283} C_VEL
LIN {X 0,Y 159.252,Z 575.903,A -85,B 0,C 180,E1 -24419.767,E2 -24419.767} C_VEL
LIN {X 0,Y 163.183,Z 567.2,A -85,B 0,C 180,E1 -24422.572,E2 -24422.572} C_VEL
LIN {X 0,Y 167.452,Z 556.831,A -85,B 0,C 180,E1 -24425.246,E2 -24425.246} C_VEL
LIN {X 0,Y 171.641,Z 545.544,A -85,B 0,C 180,E1 -24427.523,E2 -24427.523} C_VEL
LIN {X 0,Y 175.559,Z 533.201,A -85,B 0,C 180,E1 -24429.458,E2 -24429.458} C_VEL
LIN {X 0,Y 179.188,Z 519.413,A -85,B 0,C 180,E1 -24431.069,E2 -24431.069} C_VEL
LIN {X 0,Y 181.912,Z 505.549,A -85,B 0,C 180,E1 -24432.259,E2 -24432.259} C_VEL
LIN {X 0,Y 183.81,Z 491.087,A -85,B 0,C 180,E1 -24433.114,E2 -24433.114} C_VEL
LIN {X 0,Y 188.135,Z 431.724,A -85,B 0,C 180,E1 -24435.066,E2 -24435.066} C_VEL
LIN {X 0,Y 182.927,Z 421.15,A -85,B 0,C 180,E1 -24437.538,E2 -24437.538} C_VEL
LIN {X 0,Y 176.923,Z 410.587,A -85,B 0,C 180,E1 -24440.646,E2 -24440.646} C_VEL
LIN {X 0,Y 170.951,Z 401.169,A -85,B 0,C 180,E1 -24444.143,E2 -24444.143} C_VEL
LIN {X 0,Y 165.14,Z 392.917,A -85,B 0,C 180,E1 -24448.095,E2 -24448.095} C_VEL
LIN {X 0,Y 162.135,Z 388.794,A -85,B 0,C 180,E1 -24450.456,E2 -24450.456} C_VEL
LIN {X 0,Y 159.028,Z 385.232,A -85,B 0,C 180,E1 -24453.149,E2 -24453.149} C_VEL
LIN {X 0,Y 157.985,Z 383.514,A -85,B 0,C 180,E1 -24454.204,E2 -24454.204} C_VEL
LIN {X 0,Y 155.075,Z 380.684,A -85,B 0,C 180,E1 -24457.254,E2 -24457.254} C_VEL
LIN {X 0,Y 153.82,Z 378.186,A -85,B 0,C 180,E1 -24458.94,E2 -24458.94} C_VEL
LIN {X 0,Y 150.597,Z 375.796,A -85,B 0,C 180,E1 -24463.564,E2 -24463.564} C_VEL
LIN {X 0,Y 149.263,Z 372.915,A -85,B 0,C 180,E1 -24466.556,E2 -24466.556} C_VEL
LIN {X 0,Y 149.096,Z 372.303,A -85,B 0,C 180,E1 -24467.061,E2 -24467.061} C_VEL
LIN {X 0,Y 147.035,Z 371.026,A -85,B 0,C 180,E1 -24479.999,E2 -24479.999} C_VEL
LIN {X 0,Y 149.385,Z 372.397,A -85,B 0,C 180,E1 -24488.198,E2 -24488.198} C_VEL
LIN {X 0,Y 150.676,Z 375.58,A -85,B 0,C 180,E1 -24491.153,E2 -24491.153} C_VEL
LIN {X 0,Y 152.966,Z 377.719,A -85,B 0,C 180,E1 -24494.636,E2 -24494.636} C_VEL
LIN {X 0,Y 153.976,Z 378.309,A -85,B 0,C 180,E1 -24495.893,E2 -24495.893} C_VEL
LIN {X 0,Y 155.683,Z 381.364,A -85,B 0,C 180,E1 -24498.08,E2 -24498.08} C_VEL
LIN {X 0,Y 158.356,Z 383.95,A -85,B 0,C 180,E1 -24500.796,E2 -24500.796} C_VEL
LIN {X 0,Y 160.702,Z 387.379,A -85,B 0,C 180,E1 -24503.008,E2 -24503.008} C_VEL
LIN {X 0,Y 162.242,Z 389.034,A -85,B 0,C 180,E1 -24504.279,E2 -24504.279} C_VEL
LIN {X 0,Y 165.116,Z 392.872,A -85,B 0,C 180,E1 -24506.524,E2 -24506.524} C_VEL
LIN {X 0,Y 169.303,Z 398.841,A -85,B 0,C 180,E1 -24509.448,E2 -24509.448} C_VEL
LIN {X 0,Y 173.349,Z 404.838,A -85,B 0,C 180,E1 -24511.958,E2 -24511.958} C_VEL
LIN {X 0,Y 177.763,Z 413.499,A -85,B 0,C 180,E1 -24514.547,E2 -24514.547} C_VEL
LIN {X 0,Y 182.573,Z 424.146,A -85,B 0,C 180,E1 -24517.147,E2 -24517.147} C_VEL
LIN {X 0,Y 187.387,Z 436.952,A -85,B 0,C 180,E1 -24519.612,E2 -24519.612} C_VEL
LIN {X 0,Y 187.756,Z 438.116,A -85,B 0,C 180,E1 -24519.801,E2 -24519.801} C_VEL
LIN {X 0,Y 183.374,Z 498.769,A -85,B 0,C 180,E1 -24521.82,E2 -24521.82} C_VEL
LIN {X 0,Y 181.349,Z 512.657,A -85,B 0,C 180,E1 -24522.58,E2 -24522.58} C_VEL
LIN {X 0,Y 178.583,Z 526.151,A -85,B 0,C 180,E1 -24523.686,E2 -24523.686} C_VEL
LIN {X 0,Y 174.831,Z 540.218,A -85,B 0,C 180,E1 -24525.293,E2 -24525.293} C_VEL
LIN {X 0,Y 170.642,Z 552.773,A -85,B 0,C 180,E1 -24527.19,E2 -24527.19} C_VEL
LIN {X 0,Y 166.324,Z 564.352,A -85,B 0,C 180,E1 -24529.515,E2 -24529.515} C_VEL
LIN {X 0,Y 161.414,Z 575.773,A -85,B 0,C 180,E1 -24532.442,E2 -24532.442} C_VEL
LIN {X 0,Y 156.508,Z 586.036,A -85,B 0,C 180,E1 -24535.853,E2 -24535.853} C_VEL
LIN {X 0,Y 155.379,Z 588.222,A -85,B 0,C 180,E1 -24536.709,E2 -24536.709} C_VEL
LIN {X 0,Y 152.891,Z 591.951,A -85,B 0,C 180,E1 -24538.147,E2 -24538.147} C_VEL
LIN {X 0,Y 147.365,Z 597.644,A -85,B 0,C 180,E1 -24540.432,E2 -24540.432} C_VEL
LIN {X 0,Y 142.049,Z 602.762,A -85,B 0,C 180,E1 -24543.049,E2 -24543.049} C_VEL
LIN {X 0,Y 139.965,Z 605.589,A -85,B 0,C 180,E1 -24544.975,E2 -24544.975} C_VEL
LIN {X 0,Y 136.748,Z 612.001,A -85,B 0,C 180,E1 -24550.485,E2 -24550.485} C_VEL
LIN {X 0,Y 134.525,Z 617.015,A -85,B 0,C 180,E1 -24556.403,E2 -24556.403} C_VEL
LIN {X 0,Y 133.705,Z 619.78,A -85,B 0,C 180,E1 -24560.927,E2 -24560.927} C_VEL
LIN {X 0,Y 133.405,Z 622.194,A -85,B 0,C 180,E1 -24566.98,E2 -24566.98} C_VEL
LIN {X 0,Y 133.531,Z 622.885,A -85,B 0,C 180,E1 -24570,E2 -24570} C_VEL
LIN {X 0,Y 133.449,Z 623.232,A -85,B 0,C 180,E1 -24576.046,E2 -24576.046} C_VEL
LIN {X 0,Y 134.26,Z 622.251,A -85,B 0,C 180,E1 -24582.086,E2 -24582.086} C_VEL
LIN {X 0,Y 136.215,Z 619.938,A -85,B 0,C 180,E1 -24588.034,E2 -24588.034} C_VEL
LIN {X 0,Y 139.587,Z 616.241,A -85,B 0,C 180,E1 -24593.753,E2 -24593.753} C_VEL
LIN {X 0,Y 142.816,Z 612.485,A -85,B 0,C 180,E1 -24597.871,E2 -24597.871} C_VEL
LIN {X 0,Y 148.357,Z 606.041,A -85,B 0,C 180,E1 -24603.01,E2 -24603.01} C_VEL
LIN {X 0,Y 154.148,Z 598.894,A -85,B 0,C 180,E1 -24607.165,E2 -24607.165} C_VEL
LIN {X 0,Y 159.737,Z 591.429,A -85,B 0,C 180,E1 -24610.464,E2 -24610.464} C_VEL
LIN {X 0,Y 165.741,Z 582.666,A -85,B 0,C 180,E1 -24613.46,E2 -24613.46} C_VEL
LIN {X 0,Y 171.203,Z 573.616,A -85,B 0,C 180,E1 -24615.92,E2 -24615.92} C_VEL
LIN {X 0,Y 176.889,Z 563.054,A -85,B 0,C 180,E1 -24618.156,E2 -24618.156} C_VEL
LIN {X 0,Y 182.24,Z 551.563,A -85,B 0,C 180,E1 -24620.038,E2 -24620.038} C_VEL
LIN {X 0,Y 187.264,Z 538.956,A -85,B 0,C 180,E1 -24621.577,E2 -24621.577} C_VEL
LIN {X 0,Y 191.456,Z 525.942,A -85,B 0,C 180,E1 -24622.761,E2 -24622.761} C_VEL
LIN {X 0,Y 194.731,Z 512.419,A -85,B 0,C 180,E1 -24623.679,E2 -24623.679} C_VEL
LIN {X 0,Y 197.156,Z 497.937,A -85,B 0,C 180,E1 -24624.346,E2 -24624.346} C_VEL
LIN {X 0,Y 200.859,Z 455.318,A -85,B 0,C 180,E1 -24625.581,E2 -24625.581} C_VEL
LIN {X 0,Y 196.734,Z 444.688,A -85,B 0,C 180,E1 -24628.3,E2 -24628.3} C_VEL
LIN {X 0,Y 192.196,Z 434.503,A -85,B 0,C 180,E1 -24631.617,E2 -24631.617} C_VEL
LIN {X 0,Y 188.748,Z 427.516,A -85,B 0,C 180,E1 -24634.481,E2 -24634.481} C_VEL
LIN {X 0,Y 186.046,Z 422.719,A -85,B 0,C 180,E1 -24637,E2 -24637} C_VEL
LIN {X 0,Y 183.172,Z 418.45,A -85,B 0,C 180,E1 -24640.045,E2 -24640.045} C_VEL
LIN {X 0,Y 180.466,Z 414.358,A -85,B 0,C 180,E1 -24643.601,E2 -24643.601} C_VEL
LIN {X 0,Y 178.131,Z 411.196,A -85,B 0,C 180,E1 -24647.666,E2 -24647.666} C_VEL
LIN {X 0,Y 177.553,Z 409.704,A -85,B 0,C 180,E1 -24649.164,E2 -24649.164} C_VEL
LIN {X 0,Y 175.766,Z 408.082,A -85,B 0,C 180,E1 -24657.709,E2 -24657.709} C_VEL
LIN {X 0,Y 175.973,Z 408.197,A -85,B 0,C 180,E1 -24660.573,E2 -24660.573} C_VEL
LIN {X 0,Y 177.665,Z 409.788,A -85,B 0,C 180,E1 -24666.531,E2 -24666.531} C_VEL
LIN {X 0,Y 179.289,Z 413.089,A -85,B 0,C 180,E1 -24670.026,E2 -24670.026} C_VEL
LIN {X 0,Y 180.937,Z 415,A -85,B 0,C 180,E1 -24672.514,E2 -24672.514} C_VEL
LIN {X 0,Y 183.487,Z 418.849,A -85,B 0,C 180,E1 -24675.748,E2 -24675.748} C_VEL
LIN {X 0,Y 187.015,Z 424.259,A -85,B 0,C 180,E1 -24679.364,E2 -24679.364} C_VEL
LIN {X 0,Y 190.755,Z 430.102,A -85,B 0,C 180,E1 -24682.545,E2 -24682.545} C_VEL
LIN {X 0,Y 195.787,Z 438.895,A -85,B 0,C 180,E1 -24686.212,E2 -24686.212} C_VEL
LIN {X 0,Y 200.567,Z 448.184,A -85,B 0,C 180,E1 -24689.251,E2 -24689.251} C_VEL
LIN {X 0,Y 201.211,Z 449.514,A -85,B 0,C 180,E1 -24689.635,E2 -24689.635} C_VEL
LIN {X 0,Y 197.598,Z 492.334,A -85,B 0,C 180,E1 -24690.946,E2 -24690.946} C_VEL
LIN {X 0,Y 195.307,Z 506.467,A -85,B 0,C 180,E1 -24691.651,E2 -24691.651} C_VEL
LIN {X 0,Y 191.98,Z 520.397,A -85,B 0,C 180,E1 -24692.649,E2 -24692.649} C_VEL
LIN {X 0,Y 187.531,Z 534.239,A -85,B 0,C 180,E1 -24693.986,E2 -24693.986} C_VEL
LIN {X 0,Y 183.439,Z 544.801,A -85,B 0,C 180,E1 -24695.367,E2 -24695.367} C_VEL
LIN {X 0,Y 178.005,Z 556.767,A -85,B 0,C 180,E1 -24697.384,E2 -24697.384} C_VEL
LIN {X 0,Y 172.774,Z 566.372,A -85,B 0,C 180,E1 -24699.387,E2 -24699.387} C_VEL
LIN {X 0,Y 166.401,Z 577.034,A -85,B 0,C 180,E1 -24702.345,E2 -24702.345} C_VEL
LIN {X 0,Y 160.488,Z 585.801,A -85,B 0,C 180,E1 -24705.519,E2 -24705.519} C_VEL
LIN {X 0,Y 154.923,Z 593.07,A -85,B 0,C 180,E1 -24708.869,E2 -24708.869} C_VEL
LIN {X 0,Y 148.828,Z 600.452,A -85,B 0,C 180,E1 -24713.398,E2 -24713.398} C_VEL
LIN {X 0,Y 144.343,Z 605.494,A -85,B 0,C 180,E1 -24717.616,E2 -24717.616} C_VEL
LIN {X 0,Y 139.864,Z 610.236,A -85,B 0,C 180,E1 -24723.112,E2 -24723.112} C_VEL
LIN {X 0,Y 136.571,Z 613.457,A -85,B 0,C 180,E1 -24728.886,E2 -24728.886} C_VEL
LIN {X 0,Y 134.393,Z 615.27,A -85,B 0,C 180,E1 -24734.842,E2 -24734.842} C_VEL
LIN {X 0,Y 133.522,Z 615.744,A -85,B 0,C 180,E1 -24740.914,E2 -24740.914} C_VEL
LIN {X 0,Y 133.423,Z 615.487,A -85,B 0,C 180,E1 -24743.953,E2 -24743.953} C_VEL
LIN {X 0,Y 133.544,Z 614.249,A -85,B 0,C 180,E1 -24749.321,E2 -24749.321} C_VEL
LIN {X 0,Y 133.968,Z 612.753,A -85,B 0,C 180,E1 -24753.007,E2 -24753.007} C_VEL
LIN {X 0,Y 135.397,Z 609.233,A -85,B 0,C 180,E1 -24758.959,E2 -24758.959} C_VEL
LIN {X 0,Y 138.081,Z 604.225,A -85,B 0,C 180,E1 -24764.743,E2 -24764.743} C_VEL
LIN {X 0,Y 141.644,Z 597.589,A -85,B 0,C 180,E1 -24770.324,E2 -24770.324} C_VEL
LIN {X 0,Y 145.583,Z 590.19,A -85,B 0,C 180,E1 -24774.987,E2 -24774.987} C_VEL
LIN {X 0,Y 149.992,Z 582.453,A -85,B 0,C 180,E1 -24778.703,E2 -24778.703} C_VEL
LIN {X 0,Y 154.721,Z 573.146,A -85,B 0,C 180,E1 -24782.258,E2 -24782.258} C_VEL
LIN {X 0,Y 159.42,Z 562.856,A -85,B 0,C 180,E1 -24785.353,E2 -24785.353} C_VEL
LIN {X 0,Y 163.635,Z 552.78,A -85,B 0,C 180,E1 -24787.736,E2 -24787.736} C_VEL
LIN {X 0,Y 168.138,Z 540.492,A -85,B 0,C 180,E1 -24789.991,E2 -24789.991} C_VEL
LIN {X 0,Y 171.78,Z 528.687,A -85,B 0,C 180,E1 -24791.67,E2 -24791.67} C_VEL
LIN {X 0,Y 175.009,Z 515.799,A -85,B 0,C 180,E1 -24793.054,E2 -24793.054} C_VEL
LIN {X 0,Y 177.523,Z 502.005,A -85,B 0,C 180,E1 -24794.149,E2 -24794.149} C_VEL
LIN {X 0,Y 179.281,Z 487.705,A -85,B 0,C 180,E1 -24794.88,E2 -24794.88} C_VEL
LIN {X 0,Y 183.184,Z 434.18,A -85,B 0,C 180,E1 -24796.663,E2 -24796.663} C_VEL
LIN {X 0,Y 178.42,Z 424.508,A -85,B 0,C 180,E1 -24799.103,E2 -24799.103} C_VEL
LIN {X 0,Y 173.08,Z 414.935,A -85,B 0,C 180,E1 -24802.089,E2 -24802.089} C_VEL
LIN {X 0,Y 167.874,Z 406.608,A -85,B 0,C 180,E1 -24805.357,E2 -24805.357} C_VEL
LIN {X 0,Y 162.864,Z 399.157,A -85,B 0,C 180,E1 -24808.99,E2 -24808.99} C_VEL
LIN {X 0,Y 159.497,Z 394.586,A -85,B 0,C 180,E1 -24811.796,E2 -24811.796} C_VEL
LIN {X 0,Y 156.836,Z 391.176,A -85,B 0,C 180,E1 -24814.313,E2 -24814.313} C_VEL
LIN {X 0,Y 156.114,Z 390.051,A -85,B 0,C 180,E1 -24815.082,E2 -24815.082} C_VEL
LIN {X 0,Y 153.26,Z 386.964,A -85,B 0,C 180,E1 -24818.301,E2 -24818.301} C_VEL
LIN {X 0,Y 152.172,Z 384.878,A -85,B 0,C 180,E1 -24819.85,E2 -24819.85} C_VEL
LIN {X 0,Y 149.211,Z 382.393,A -85,B 0,C 180,E1 -24824.46,E2 -24824.46} C_VEL
LIN {X 0,Y 147.953,Z 379.292,A -85,B 0,C 180,E1 -24827.657,E2 -24827.657} C_VEL
LIN {X 0,Y 146.168,Z 378.08,A -85,B 0,C 180,E1 -24839.999,E2 -24839.999} C_VEL
LIN {X 0,Y 148.235,Z 379.51,A -85,B 0,C 180,E1 -24847.662,E2 -24847.662} C_VEL
LIN {X 0,Y 149.717,Z 382.805,A -85,B 0,C 180,E1 -24851.084,E2 -24851.084} C_VEL
LIN {X 0,Y 152.474,Z 385.202,A -85,B 0,C 180,E1 -24855.197,E2 -24855.197} C_VEL
LIN {X 0,Y 154.602,Z 388.619,A -85,B 0,C 180,E1 -24857.954,E2 -24857.954} C_VEL
LIN {X 0,Y 156.575,Z 390.627,A -85,B 0,C 180,E1 -24860.034,E2 -24860.034} C_VEL
LIN {X 0,Y 159.253,Z 394.333,A -85,B 0,C 180,E1 -24862.629,E2 -24862.629} C_VEL
LIN {X 0,Y 160.496,Z 396.018,A -85,B 0,C 180,E1 -24863.722,E2 -24863.722} C_VEL
LIN {X 0,Y 163.677,Z 400.376,A -85,B 0,C 180,E1 -24866.282,E2 -24866.282} C_VEL
LIN {X 0,Y 167.078,Z 405.404,A -85,B 0,C 180,E1 -24868.742,E2 -24868.742} C_VEL
LIN {X 0,Y 170.434,Z 410.593,A -85,B 0,C 180,E1 -24870.941,E2 -24870.941} C_VEL
LIN {X 0,Y 174.382,Z 418.692,A -85,B 0,C 180,E1 -24873.412,E2 -24873.412} C_VEL
LIN {X 0,Y 178.781,Z 428.852,A -85,B 0,C 180,E1 -24875.958,E2 -24875.958} C_VEL
LIN {X 0,Y 182.88,Z 440.099,A -85,B 0,C 180,E1 -24878.213,E2 -24878.213} C_VEL
LIN {X 0,Y 178.586,Z 497.996,A -85,B 0,C 180,E1 -24880.163,E2 -24880.163} C_VEL
LIN {X 0,Y 176.471,Z 512.214,A -85,B 0,C 180,E1 -24880.936,E2 -24880.936} C_VEL
LIN {X 0,Y 173.454,Z 526.338,A -85,B 0,C 180,E1 -24882.099,E2 -24882.099} C_VEL
LIN {X 0,Y 169.825,Z 539.43,A -85,B 0,C 180,E1 -24883.596,E2 -24883.596} C_VEL
LIN {X 0,Y 165.483,Z 552.1,A -85,B 0,C 180,E1 -24885.513,E2 -24885.513} C_VEL
LIN {X 0,Y 161.061,Z 563.537,A -85,B 0,C 180,E1 -24887.817,E2 -24887.817} C_VEL
LIN {X 0,Y 156.716,Z 573.284,A -85,B 0,C 180,E1 -24890.279,E2 -24890.279} C_VEL
LIN {X 0,Y 151.468,Z 583.973,A -85,B 0,C 180,E1 -24893.73,E2 -24893.73} C_VEL
LIN {X 0,Y 146.821,Z 592.792,A -85,B 0,C 180,E1 -24897.417,E2 -24897.417} C_VEL
LIN {X 0,Y 142.24,Z 601.251,A -85,B 0,C 180,E1 -24902.005,E2 -24902.005} C_VEL
LIN {X 0,Y 139.965,Z 605.589,A -85,B 0,C 180,E1 -24904.975,E2 -24904.975} C_VEL
LIN {X 0,Y 137.982,Z 608.286,A -85,B 0,C 180,E1 -24906.999,E2 -24906.999} C_VEL
LIN {X 0,Y 131.254,Z 613.56,A -85,B 0,C 180,E1 -24911.672,E2 -24911.672} C_VEL
LIN {X 0,Y 128.166,Z 616.064,A -85,B 0,C 180,E1 -24914.7,E2 -24914.7} C_VEL
LIN {X 0,Y 127.409,Z 617.192,A -85,B 0,C 180,E1 -24916.358,E2 -24916.358} C_VEL
LIN {X 0,Y 126.657,Z 619.518,A -85,B 0,C 180,E1 -24920.418,E2 -24920.418} C_VEL
LIN {X 0,Y 126.39,Z 620.913,A -85,B 0,C 180,E1 -24923.615,E2 -24923.615} C_VEL
LIN {X 0,Y 126.427,Z 622.663,A -85,B 0,C 180,E1 -24930,E2 -24930} C_VEL
LIN {X 0,Y 126.389,Z 623.036,A -85,B 0,C 180,E1 -24936.385,E2 -24936.385} C_VEL
LIN {X 0,Y 127.297,Z 622.082,A -85,B 0,C 180,E1 -24942.758,E2 -24942.758} C_VEL
LIN {X 0,Y 129.455,Z 619.795,A -85,B 0,C 180,E1 -24949.01,E2 -24949.01} C_VEL
LIN {X 0,Y 133.077,Z 616.126,A -85,B 0,C 180,E1 -24954.992,E2 -24954.992} C_VEL
LIN {X 0,Y 136.544,Z 612.4,A -85,B 0,C 180,E1 -24959.272,E2 -24959.272} C_VEL
LIN {X 0,Y 142.428,Z 605.988,A -85,B 0,C 180,E1 -24964.574,E2 -24964.574} C_VEL
LIN {X 0,Y 148.515,Z 598.875,A -85,B 0,C 180,E1 -24968.831,E2 -24968.831} C_VEL
LIN {X 0,Y 155.456,Z 590.095,A -85,B 0,C 180,E1 -24972.698,E2 -24972.698} C_VEL
LIN {X 0,Y 162.103,Z 580.556,A -85,B 0,C 180,E1 -24975.874,E2 -24975.874} C_VEL
LIN {X 0,Y 168.648,Z 569.796,A -85,B 0,C 180,E1 -24978.6,E2 -24978.6} C_VEL
LIN {X 0,Y 174.663,Z 558.461,A -85,B 0,C 180,E1 -24980.767,E2 -24980.767} C_VEL
LIN {X 0,Y 179.719,Z 547.51,A -85,B 0,C 180,E1 -24982.363,E2 -24982.363} C_VEL
LIN {X 0,Y 184.273,Z 535.785,A -85,B 0,C 180,E1 -24983.677,E2 -24983.677} C_VEL
LIN {X 0,Y 188.563,Z 521.777,A -85,B 0,C 180,E1 -24984.85,E2 -24984.85} C_VEL
LIN {X 0,Y 191.805,Z 507.329,A -85,B 0,C 180,E1 -24985.704,E2 -24985.704} C_VEL
LIN {X 0,Y 193.883,Z 492.849,A -85,B 0,C 180,E1 -24986.269,E2 -24986.269} C_VEL
LIN {X 0,Y 196.91,Z 458.067,A -85,B 0,C 180,E1 -24987.256,E2 -24987.256} C_VEL
LIN {X 0,Y 193.396,Z 448.782,A -85,B 0,C 180,E1 -24989.777,E2 -24989.777} C_VEL
LIN {X 0,Y 189.506,Z 439.624,A -85,B 0,C 180,E1 -24992.866,E2 -24992.866} C_VEL
LIN {X 0,Y 186.065,Z 432.323,A -85,B 0,C 180,E1 -24995.984,E2 -24995.984} C_VEL
LIN {X 0,Y 184.055,Z 428.833,A -85,B 0,C 180,E1 -24997.996,E2 -24997.996} C_VEL
LIN {X 0,Y 181.558,Z 424.949,A -85,B 0,C 180,E1 -25000.826,E2 -25000.826} C_VEL
LIN {X 0,Y 179.142,Z 421.109,A -85,B 0,C 180,E1 -25004.207,E2 -25004.207} C_VEL
LIN {X 0,Y 176.923,Z 417.836,A -85,B 0,C 180,E1 -25008.384,E2 -25008.384} C_VEL
LIN {X 0,Y 176.463,Z 416.618,A -85,B 0,C 180,E1 -25009.676,E2 -25009.676} C_VEL
LIN {X 0,Y 174.898,Z 415.143,A -85,B 0,C 180,E1 -25017.698,E2 -25017.698} C_VEL
LIN {X 0,Y 175.104,Z 415.265,A -85,B 0,C 180,E1 -25020.576,E2 -25020.576} C_VEL
LIN {X 0,Y 176.609,Z 416.803,A -85,B 0,C 180,E1 -25026.14,E2 -25026.14} C_VEL
LIN {X 0,Y 178.49,Z 420.43,A -85,B 0,C 180,E1 -25030.208,E2 -25030.208} C_VEL
LIN {X 0,Y 179.604,Z 421.804,A -85,B 0,C 180,E1 -25031.939,E2 -25031.939} C_VEL
LIN {X 0,Y 182.719,Z 426.773,A -85,B 0,C 180,E1 -25035.993,E2 -25035.993} C_VEL
LIN {X 0,Y 185.408,Z 431.027,A -85,B 0,C 180,E1 -25038.805,E2 -25038.805} C_VEL
LIN {X 0,Y 188.821,Z 436.644,A -85,B 0,C 180,E1 -25041.852,E2 -25041.852} C_VEL
LIN {X 0,Y 193.452,Z 445.066,A -85,B 0,C 180,E1 -25045.403,E2 -25045.403} C_VEL
LIN {X 0,Y 197.316,Z 452.879,A -85,B 0,C 180,E1 -25048.017,E2 -25048.017} C_VEL
LIN {X 0,Y 193.781,Z 492.494,A -85,B 0,C 180,E1 -25049.2,E2 -25049.2} C_VEL
LIN {X 0,Y 191.494,Z 506.309,A -85,B 0,C 180,E1 -25049.88,E2 -25049.88} C_VEL
LIN {X 0,Y 188.233,Z 519.763,A -85,B 0,C 180,E1 -25050.823,E2 -25050.823} C_VEL
LIN {X 0,Y 184.293,Z 532.008,A -85,B 0,C 180,E1 -25051.95,E2 -25051.95} C_VEL
LIN {X 0,Y 179.9,Z 543.217,A -85,B 0,C 180,E1 -25053.303,E2 -25053.303} C_VEL
LIN {X 0,Y 174.355,Z 555.354,A -85,B 0,C 180,E1 -25055.288,E2 -25055.288} C_VEL
LIN {X 0,Y 168.332,Z 566.213,A -85,B 0,C 180,E1 -25057.507,E2 -25057.507} C_VEL
LIN {X 0,Y 162.718,Z 575.299,A -85,B 0,C 180,E1 -25059.947,E2 -25059.947} C_VEL
LIN {X 0,Y 156.456,Z 584.394,A -85,B 0,C 180,E1 -25063.117,E2 -25063.117} C_VEL
LIN {X 0,Y 149.575,Z 593.066,A -85,B 0,C 180,E1 -25067.054,E2 -25067.054} C_VEL
LIN {X 0,Y 144.313,Z 599.135,A -85,B 0,C 180,E1 -25070.721,E2 -25070.721} C_VEL
LIN {X 0,Y 139.695,Z 604.144,A -85,B 0,C 180,E1 -25074.65,E2 -25074.65} C_VEL
LIN {X 0,Y 134.558,Z 609.282,A -85,B 0,C 180,E1 -25080.252,E2 -25080.252} C_VEL
LIN {X 0,Y 130.828,Z 612.772,A -85,B 0,C 180,E1 -25085.958,E2 -25085.958} C_VEL
LIN {X 0,Y 128.56,Z 614.698,A -85,B 0,C 180,E1 -25090.852,E2 -25090.852} C_VEL
LIN {X 0,Y 126.816,Z 615.868,A -85,B 0,C 180,E1 -25097.192,E2 -25097.192} C_VEL
LIN {X 0,Y 126.318,Z 615.712,A -85,B 0,C 180,E1 -25103.611,E2 -25103.611} C_VEL
LIN {X 0,Y 126.372,Z 615.143,A -85,B 0,C 180,E1 -25106.812,E2 -25106.812} C_VEL
LIN {X 0,Y 126.88,Z 613.022,A -85,B 0,C 180,E1 -25113.175,E2 -25113.175} C_VEL
LIN {X 0,Y 128.407,Z 609.531,A -85,B 0,C 180,E1 -25119.451,E2 -25119.451} C_VEL
LIN {X 0,Y 131.26,Z 604.556,A -85,B 0,C 180,E1 -25125.528,E2 -25125.528} C_VEL
LIN {X 0,Y 135.019,Z 597.962,A -85,B 0,C 180,E1 -25131.368,E2 -25131.368} C_VEL
LIN {X 0,Y 139.201,Z 590.615,A -85,B 0,C 180,E1 -25136.217,E2 -25136.217} C_VEL
LIN {X 0,Y 143.825,Z 582.912,A -85,B 0,C 180,E1 -25140.057,E2 -25140.057} C_VEL
LIN {X 0,Y 148.795,Z 573.667,A -85,B 0,C 180,E1 -25143.71,E2 -25143.71} C_VEL
LIN {X 0,Y 153.716,Z 563.448,A -85,B 0,C 180,E1 -25146.876,E2 -25146.876} C_VEL
LIN {X 0,Y 158.089,Z 553.433,A -85,B 0,C 180,E1 -25149.309,E2 -25149.309} C_VEL
LIN {X 0,Y 162.788,Z 541.274,A -85,B 0,C 180,E1 -25151.589,E2 -25151.589} C_VEL
LIN {X 0,Y 166.586,Z 529.605,A -85,B 0,C 180,E1 -25153.28,E2 -25153.28} C_VEL
LIN {X 0,Y 170.208,Z 515.66,A -85,B 0,C 180,E1 -25154.791,E2 -25154.791} C_VEL
LIN {X 0,Y 172.826,Z 501.727,A -85,B 0,C 180,E1 -25155.89,E2 -25155.89} C_VEL
LIN {X 0,Y 174.617,Z 487.497,A -85,B 0,C 180,E1 -25156.608,E2 -25156.608} C_VEL
LIN {X 0,Y 178.469,Z 436.969,A -85,B 0,C 180,E1 -25158.293,E2 -25158.293} C_VEL
LIN {X 0,Y 173.579,Z 426.977,A -85,B 0,C 180,E1 -25161.02,E2 -25161.02} C_VEL
LIN {X 0,Y 169.04,Z 418.77,A -85,B 0,C 180,E1 -25163.795,E2 -25163.795} C_VEL
LIN {X 0,Y 164.092,Z 410.796,A -85,B 0,C 180,E1 -25167.19,E2 -25167.19} C_VEL
LIN {X 0,Y 159.98,Z 404.603,A -85,B 0,C 180,E1 -25170.441,E2 -25170.441} C_VEL
LIN {X 0,Y 157.368,Z 400.862,A -85,B 0,C 180,E1 -25172.791,E2 -25172.791} C_VEL
LIN {X 0,Y 154.624,Z 396.942,A -85,B 0,C 180,E1 -25175.611,E2 -25175.611} C_VEL
LIN {X 0,Y 151.559,Z 393.341,A -85,B 0,C 180,E1 -25179.285,E2 -25179.285} C_VEL
LIN {X 0,Y 150.68,Z 391.648,A -85,B 0,C 180,E1 -25180.618,E2 -25180.618} C_VEL
LIN {X 0,Y 147.863,Z 388.976,A -85,B 0,C 180,E1 -25185.373,E2 -25185.373} C_VEL
LIN {X 0,Y 146.826,Z 386.245,A -85,B 0,C 180,E1 -25188.275,E2 -25188.275} C_VEL
LIN {X 0,Y 145.298,Z 385.147,A -85,B 0,C 180,E1 -25199.999,E2 -25199.999} C_VEL
LIN {X 0,Y 147.086,Z 386.424,A -85,B 0,C 180,E1 -25207.032,E2 -25207.032} C_VEL
LIN {X 0,Y 148.7,Z 389.907,A -85,B 0,C 180,E1 -25210.897,E2 -25210.897} C_VEL
LIN {X 0,Y 151.006,Z 392.003,A -85,B 0,C 180,E1 -25214.486,E2 -25214.486} C_VEL
LIN {X 0,Y 153.123,Z 395.385,A -85,B 0,C 180,E1 -25217.357,E2 -25217.357} C_VEL
LIN {X 0,Y 154.793,Z 397.216,A -85,B 0,C 180,E1 -25219.218,E2 -25219.218} C_VEL
LIN {X 0,Y 157.647,Z 401.112,A -85,B 0,C 180,E1 -25222.095,E2 -25222.095} C_VEL
LIN {X 0,Y 161.677,Z 407.073,A -85,B 0,C 180,E1 -25225.592,E2 -25225.592} C_VEL
LIN {X 0,Y 165.807,Z 413.265,A -85,B 0,C 180,E1 -25228.663,E2 -25228.663} C_VEL
LIN {X 0,Y 168.831,Z 418.9,A -85,B 0,C 180,E1 -25230.746,E2 -25230.746} C_VEL
LIN {X 0,Y 173.64,Z 429.925,A -85,B 0,C 180,E1 -25233.847,E2 -25233.847} C_VEL
LIN {X 0,Y 177.493,Z 440.42,A -85,B 0,C 180,E1 -25236.172,E2 -25236.172} C_VEL
LIN {X 0,Y 178.166,Z 442.398,A -85,B 0,C 180,E1 -25236.566,E2 -25236.566} C_VEL
LIN {X 0,Y 173.825,Z 498.131,A -85,B 0,C 180,E1 -25238.454,E2 -25238.454} C_VEL
LIN {X 0,Y 171.583,Z 512.534,A -85,B 0,C 180,E1 -25239.249,E2 -25239.249} C_VEL
LIN {X 0,Y 168.467,Z 526.524,A -85,B 0,C 180,E1 -25240.417,E2 -25240.417} C_VEL
LIN {X 0,Y 164.431,Z 540.422,A -85,B 0,C 180,E1 -25242.044,E2 -25242.044} C_VEL
LIN {X 0,Y 159.918,Z 552.861,A -85,B 0,C 180,E1 -25243.975,E2 -25243.975} C_VEL
LIN {X 0,Y 155.458,Z 563.799,A -85,B 0,C 180,E1 -25246.242,E2 -25246.242} C_VEL
LIN {X 0,Y 151.311,Z 572.76,A -85,B 0,C 180,E1 -25248.557,E2 -25248.557} C_VEL
LIN {X 0,Y 145.767,Z 583.501,A -85,B 0,C 180,E1 -25252.068,E2 -25252.068} C_VEL
LIN {X 0,Y 140.83,Z 592.364,A -85,B 0,C 180,E1 -25255.846,E2 -25255.846} C_VEL
LIN {X 0,Y 135.951,Z 600.862,A -85,B 0,C 180,E1 -25260.587,E2 -25260.587} C_VEL
LIN {X 0,Y 132.655,Z 606.792,A -85,B 0,C 180,E1 -25264.923,E2 -25264.923} C_VEL
LIN {X 0,Y 129.292,Z 613.122,A -85,B 0,C 180,E1 -25270.965,E2 -25270.965} C_VEL
LIN {X 0,Y 127.409,Z 617.192,A -85,B 0,C 180,E1 -25276.358,E2 -25276.358} C_VEL
LIN {X 0,Y 126.305,Z 618.74,A -85,B 0,C 180,E1 -25278.88,E2 -25278.88} C_VEL
LIN {X 0,Y 123.141,Z 620.745,A -85,B 0,C 180,E1 -25283.085,E2 -25283.085} C_VEL
LIN {X 0,Y 119.73,Z 622.217,A -85,B 0,C 180,E1 -25288.472,E2 -25288.472} C_VEL
LIN {X 0,Y 119.299,Z 622.482,A -85,B 0,C 180,E1 -25290.37,E2 -25290.37} C_VEL
LIN {X 0,Y 119.304,Z 622.841,A -85,B 0,C 180,E1 -25296.766,E2 -25296.766} C_VEL
LIN {X 0,Y 120.344,Z 621.912,A -85,B 0,C 180,E1 -25303.509,E2 -25303.509} C_VEL
LIN {X 0,Y 122.741,Z 619.653,A -85,B 0,C 180,E1 -25310.094,E2 -25310.094} C_VEL
LIN {X 0,Y 126.632,Z 616.011,A -85,B 0,C 180,E1 -25316.359,E2 -25316.359} C_VEL
LIN {X 0,Y 130.362,Z 612.314,A -85,B 0,C 180,E1 -25320.808,E2 -25320.808} C_VEL
LIN {X 0,Y 136.6,Z 605.935,A -85,B 0,C 180,E1 -25326.276,E2 -25326.276} C_VEL
LIN {X 0,Y 143.037,Z 598.857,A -85,B 0,C 180,E1 -25330.62,E2 -25330.62} C_VEL
LIN {X 0,Y 150.307,Z 590.116,A -85,B 0,C 180,E1 -25334.537,E2 -25334.537} C_VEL
LIN {X 0,Y 157.559,Z 580.174,A -85,B 0,C 180,E1 -25337.865,E2 -25337.865} C_VEL
LIN {X 0,Y 164.646,Z 568.881,A -85,B 0,C 180,E1 -25340.686,E2 -25340.686} C_VEL
LIN {X 0,Y 170.942,Z 557.398,A -85,B 0,C 180,E1 -25342.805,E2 -25342.805} C_VEL
LIN {X 0,Y 176.171,Z 546.255,A -85,B 0,C 180,E1 -25344.373,E2 -25344.373} C_VEL
LIN {X 0,Y 180.832,Z 534.272,A -85,B 0,C 180,E1 -25345.678,E2 -25345.678} C_VEL
LIN {X 0,Y 184.917,Z 521.147,A -85,B 0,C 180,E1 -25346.735,E2 -25346.735} C_VEL
LIN {X 0,Y 188.23,Z 506.689,A -85,B 0,C 180,E1 -25347.561,E2 -25347.561} C_VEL
LIN {X 0,Y 190.382,Z 491.912,A -85,B 0,C 180,E1 -25348.109,E2 -25348.109} C_VEL
LIN {X 0,Y 193.128,Z 460.903,A -85,B 0,C 180,E1 -25348.996,E2 -25348.996} C_VEL
LIN {X 0,Y 189.67,Z 451.566,A -85,B 0,C 180,E1 -25351.733,E2 -25351.733} C_VEL
LIN {X 0,Y 186.082,Z 442.912,A -85,B 0,C 180,E1 -25354.917,E2 -25354.917} C_VEL
LIN {X 0,Y 183.167,Z 436.626,A -85,B 0,C 180,E1 -25357.884,E2 -25357.884} C_VEL
LIN {X 0,Y 180.089,Z 431.578,A -85,B 0,C 180,E1 -25361.482,E2 -25361.482} C_VEL
LIN {X 0,Y 177.777,Z 427.78,A -85,B 0,C 180,E1 -25364.926,E2 -25364.926} C_VEL
LIN {X 0,Y 175.713,Z 424.401,A -85,B 0,C 180,E1 -25369.195,E2 -25369.195} C_VEL
LIN {X 0,Y 175.413,Z 423.555,A -85,B 0,C 180,E1 -25370.124,E2 -25370.124} C_VEL
LIN {X 0,Y 174.032,Z 422.192,A -85,B 0,C 180,E1 -25377.686,E2 -25377.686} C_VEL
LIN {X 0,Y 174.29,Z 422.435,A -85,B 0,C 180,E1 -25380.989,E2 -25380.989} C_VEL
LIN {X 0,Y 175.564,Z 423.803,A -85,B 0,C 180,E1 -25385.744,E2 -25385.744} C_VEL
LIN {X 0,Y 177.29,Z 427.247,A -85,B 0,C 180,E1 -25389.7,E2 -25389.7} C_VEL
LIN {X 0,Y 178.298,Z 428.609,A -85,B 0,C 180,E1 -25391.367,E2 -25391.367} C_VEL
LIN {X 0,Y 181.063,Z 433.204,A -85,B 0,C 180,E1 -25395.19,E2 -25395.19} C_VEL
LIN {X 0,Y 183.762,Z 437.686,A -85,B 0,C 180,E1 -25398.177,E2 -25398.177} C_VEL
LIN {X 0,Y 186.632,Z 442.633,A -85,B 0,C 180,E1 -25400.89,E2 -25400.89} C_VEL
LIN {X 0,Y 190.699,Z 450.328,A -85,B 0,C 180,E1 -25404.227,E2 -25404.227} C_VEL
LIN {X 0,Y 193.496,Z 456.135,A -85,B 0,C 180,E1 -25406.279,E2 -25406.279} C_VEL
LIN {X 0,Y 190.174,Z 492.511,A -85,B 0,C 180,E1 -25407.379,E2 -25407.379} C_VEL
LIN {X 0,Y 187.729,Z 506.73,A -85,B 0,C 180,E1 -25408.065,E2 -25408.065} C_VEL
LIN {X 0,Y 184.326,Z 520.272,A -85,B 0,C 180,E1 -25409.006,E2 -25409.006} C_VEL
LIN {X 0,Y 179.941,Z 533.34,A -85,B 0,C 180,E1 -25410.214,E2 -25410.214} C_VEL
LIN {X 0,Y 175.604,Z 543.918,A -85,B 0,C 180,E1 -25411.499,E2 -25411.499} C_VEL
LIN {X 0,Y 169.686,Z 556.303,A -85,B 0,C 180,E1 -25413.536,E2 -25413.536} C_VEL
LIN {X 0,Y 164.065,Z 566.055,A -85,B 0,C 180,E1 -25415.521,E2 -25415.521} C_VEL
LIN {X 0,Y 158.184,Z 575.2,A -85,B 0,C 180,E1 -25417.944,E2 -25417.944} C_VEL
LIN {X 0,Y 151.6,Z 584.379,A -85,B 0,C 180,E1 -25421.144,E2 -25421.144} C_VEL
LIN {X 0,Y 144.376,Z 593.062,A -85,B 0,C 180,E1 -25425.102,E2 -25425.102} C_VEL
LIN {X 0,Y 138.806,Z 599.171,A -85,B 0,C 180,E1 -25428.836,E2 -25428.836} C_VEL
LIN {X 0,Y 133.885,Z 604.215,A -85,B 0,C 180,E1 -25432.867,E2 -25432.867} C_VEL
LIN {X 0,Y 128.344,Z 609.387,A -85,B 0,C 180,E1 -25438.653,E2 -25438.653} C_VEL
LIN {X 0,Y 124.023,Z 613.111,A -85,B 0,C 180,E1 -25445.052,E2 -25445.052} C_VEL
LIN {X 0,Y 121.784,Z 614.86,A -85,B 0,C 180,E1 -25449.741,E2 -25449.741} C_VEL
LIN {X 0,Y 119.829,Z 616.065,A -85,B 0,C 180,E1 -25456.432,E2 -25456.432} C_VEL
LIN {X 0,Y 119.228,Z 615.937,A -85,B 0,C 180,E1 -25463.229,E2 -25463.229} C_VEL
LIN {X 0,Y 119.275,Z 615.382,A -85,B 0,C 180,E1 -25466.622,E2 -25466.622} C_VEL
LIN {X 0,Y 119.813,Z 613.289,A -85,B 0,C 180,E1 -25473.363,E2 -25473.363} C_VEL
LIN {X 0,Y 121.432,Z 609.83,A -85,B 0,C 180,E1 -25479.999,E2 -25479.999} C_VEL
LIN {X 0,Y 124.457,Z 604.888,A -85,B 0,C 180,E1 -25486.4,E2 -25486.4} C_VEL
LIN {X 0,Y 128.46,Z 598.329,A -85,B 0,C 180,E1 -25492.518,E2 -25492.518} C_VEL
LIN {X 0,Y 132.894,Z 591.032,A -85,B 0,C 180,E1 -25497.564,E2 -25497.564} C_VEL
LIN {X 0,Y 138.618,Z 581.928,A -85,B 0,C 180,E1 -25502.165,E2 -25502.165} C_VEL
LIN {X 0,Y 143.893,Z 572.432,A -85,B 0,C 180,E1 -25505.881,E2 -25505.881} C_VEL
LIN {X 0,Y 149.127,Z 561.917,A -85,B 0,C 180,E1 -25509.075,E2 -25509.075} C_VEL
LIN {X 0,Y 153.24,Z 552.849,A -85,B 0,C 180,E1 -25511.245,E2 -25511.245} C_VEL
LIN {X 0,Y 158.154,Z 540.479,A -85,B 0,C 180,E1 -25513.534,E2 -25513.534} C_VEL
LIN {X 0,Y 162.094,Z 528.568,A -85,B 0,C 180,E1 -25515.234,E2 -25515.234} C_VEL
LIN {X 0,Y 165.578,Z 515.52,A -85,B 0,C 180,E1 -25516.625,E2 -25516.625} C_VEL
LIN {X 0,Y 168.301,Z 501.448,A -85,B 0,C 180,E1 -25517.724,E2 -25517.724} C_VEL
LIN {X 0,Y 170.067,Z 487.8,A -85,B 0,C 180,E1 -25518.411,E2 -25518.411} C_VEL
LIN {X 0,Y 173.922,Z 439.772,A -85,B 0,C 180,E1 -25520,E2 -25520} C_VEL
LIN {X 0,Y 168.932,Z 429.558,A -85,B 0,C 180,E1 -25523.042,E2 -25523.042} C_VEL
LIN {X 0,Y 164.406,Z 421.365,A -85,B 0,C 180,E1 -25526.113,E2 -25526.113} C_VEL
LIN {X 0,Y 159.552,Z 413.53,A -85,B 0,C 180,E1 -25529.877,E2 -25529.877} C_VEL
LIN {X 0,Y 155.761,Z 407.614,A -85,B 0,C 180,E1 -25533.359,E2 -25533.359} C_VEL
LIN {X 0,Y 152.938,Z 403.641,A -85,B 0,C 180,E1 -25536.381,E2 -25536.381} C_VEL
LIN {X 0,Y 149.774,Z 399.453,A -85,B 0,C 180,E1 -25540.497,E2 -25540.497} C_VEL
LIN {X 0,Y 149.346,Z 398.502,A -85,B 0,C 180,E1 -25541.212,E2 -25541.212} C_VEL
LIN {X 0,Y 146.623,Z 395.688,A -85,B 0,C 180,E1 -25546.132,E2 -25546.132} C_VEL
LIN {X 0,Y 145.724,Z 393.211,A -85,B 0,C 180,E1 -25548.876,E2 -25548.876} C_VEL
LIN {X 0,Y 144.429,Z 392.214,A -85,B 0,C 180,E1 -25559.999,E2 -25559.999} C_VEL
LIN {X 0,Y 146.017,Z 393.542,A -85,B 0,C 180,E1 -25566.607,E2 -25566.607} C_VEL
LIN {X 0,Y 147.558,Z 396.835,A -85,B 0,C 180,E1 -25570.461,E2 -25570.461} C_VEL
LIN {X 0,Y 149.648,Z 398.989,A -85,B 0,C 180,E1 -25573.905,E2 -25573.905} C_VEL
LIN {X 0,Y 152.087,Z 402.616,A -85,B 0,C 180,E1 -25577.262,E2 -25577.262} C_VEL
LIN {X 0,Y 153.125,Z 403.945,A -85,B 0,C 180,E1 -25578.48,E2 -25578.48} C_VEL
LIN {X 0,Y 156.332,Z 408.624,A -85,B 0,C 180,E1 -25581.856,E2 -25581.856} C_VEL
LIN {X 0,Y 159.416,Z 413.255,A -85,B 0,C 180,E1 -25584.639,E2 -25584.639} C_VEL
LIN {X 0,Y 163.628,Z 419.991,A -85,B 0,C 180,E1 -25587.955,E2 -25587.955} C_VEL
LIN {X 0,Y 166.718,Z 426.389,A -85,B 0,C 180,E1 -25590.213,E2 -25590.213} C_VEL
LIN {X 0,Y 171.156,Z 437.51,A -85,B 0,C 180,E1 -25593.241,E2 -25593.241} C_VEL
LIN {X 0,Y 173.607,Z 444.733,A -85,B 0,C 180,E1 -25594.833,E2 -25594.833} C_VEL
LIN {X 0,Y 169.327,Z 497.691,A -85,B 0,C 180,E1 -25596.633,E2 -25596.633} C_VEL
LIN {X 0,Y 167.02,Z 512.092,A -85,B 0,C 180,E1 -25597.416,E2 -25597.416} C_VEL
LIN {X 0,Y 163.911,Z 525.569,A -85,B 0,C 180,E1 -25598.509,E2 -25598.509} C_VEL
LIN {X 0,Y 160.304,Z 537.852,A -85,B 0,C 180,E1 -25599.894,E2 -25599.894} C_VEL
LIN {X 0,Y 155.625,Z 550.751,A -85,B 0,C 180,E1 -25601.829,E2 -25601.829} C_VEL
LIN {X 0,Y 150.676,Z 562.483,A -85,B 0,C 180,E1 -25604.183,E2 -25604.183} C_VEL
LIN {X 0,Y 145.978,Z 572.368,A -85,B 0,C 180,E1 -25606.745,E2 -25606.745} C_VEL
LIN {X 0,Y 140.205,Z 583.029,A -85,B 0,C 180,E1 -25610.274,E2 -25610.274} C_VEL
LIN {X 0,Y 134.965,Z 591.936,A -85,B 0,C 180,E1 -25614.139,E2 -25614.139} C_VEL
LIN {X 0,Y 129.763,Z 600.474,A -85,B 0,C 180,E1 -25619.034,E2 -25619.034} C_VEL
LIN {X 0,Y 126.182,Z 606.438,A -85,B 0,C 180,E1 -25623.54,E2 -25623.54} C_VEL
LIN {X 0,Y 123.351,Z 611.36,A -85,B 0,C 180,E1 -25628.263,E2 -25628.263} C_VEL
LIN {X 0,Y 120.672,Z 616.433,A -85,B 0,C 180,E1 -25634.806,E2 -25634.806} C_VEL
LIN {X 0,Y 119.632,Z 619.255,A -85,B 0,C 180,E1 -25639.849,E2 -25639.849} C_VEL
LIN {X 0,Y 119.219,Z 621.725,A -85,B 0,C 180,E1 -25646.621,E2 -25646.621} C_VEL
LIN {X 0,Y 119.299,Z 622.482,A -85,B 0,C 180,E1 -25650.37,E2 -25650.37} C_VEL
LIN {X 0,Y 118.496,Z 622.784,A -85,B 0,C 180,E1 -25653.187,E2 -25653.187} C_VEL
LIN {X 0,Y 115.811,Z 622.695,A -85,B 0,C 180,E1 -25657.859,E2 -25657.859} C_VEL
LIN {X 0,Y 113.929,Z 622.239,A -85,B 0,C 180,E1 -25661.733,E2 -25661.733} C_VEL
LIN {X 0,Y 113.566,Z 621.658,A -85,B 0,C 180,E1 -25664.714,E2 -25664.714} C_VEL
LIN {X 0,Y 113.761,Z 621.381,A -85,B 0,C 180,E1 -25665.702,E2 -25665.702} C_VEL
LIN {X 0,Y 116.076,Z 619.511,A -85,B 0,C 180,E1 -25671.302,E2 -25671.302} C_VEL
LIN {X 0,Y 120.26,Z 615.896,A -85,B 0,C 180,E1 -25677.874,E2 -25677.874} C_VEL
LIN {X 0,Y 124.269,Z 612.228,A -85,B 0,C 180,E1 -25682.498,E2 -25682.498} C_VEL
LIN {X 0,Y 130.907,Z 605.882,A -85,B 0,C 180,E1 -25688.127,E2 -25688.127} C_VEL
LIN {X 0,Y 137.714,Z 598.841,A -85,B 0,C 180,E1 -25692.547,E2 -25692.547} C_VEL
LIN {X 0,Y 145.317,Z 590.14,A -85,B 0,C 180,E1 -25696.507,E2 -25696.507} C_VEL
LIN {X 0,Y 152.459,Z 580.82,A -85,B 0,C 180,E1 -25699.667,E2 -25699.667} C_VEL
LIN {X 0,Y 159.608,Z 570.079,A -85,B 0,C 180,E1 -25702.429,E2 -25702.429} C_VEL
LIN {X 0,Y 166.069,Z 558.912,A -85,B 0,C 180,E1 -25704.554,E2 -25704.554} C_VEL
LIN {X 0,Y 171.454,Z 548.107,A -85,B 0,C 180,E1 -25706.106,E2 -25706.106} C_VEL
LIN {X 0,Y 176.257,Z 536.584,A -85,B 0,C 180,E1 -25707.388,E2 -25707.388} C_VEL
LIN {X 0,Y 180.804,Z 523.074,A -85,B 0,C 180,E1 -25708.511,E2 -25708.511} C_VEL
LIN {X 0,Y 184.349,Z 508.727,A -85,B 0,C 180,E1 -25709.36,E2 -25709.36} C_VEL
LIN {X 0,Y 186.579,Z 495.278,A -85,B 0,C 180,E1 -25709.897,E2 -25709.897} C_VEL
LIN {X 0,Y 189.524,Z 463.815,A -85,B 0,C 180,E1 -25710.804,E2 -25710.804} C_VEL
LIN {X 0,Y 186.219,Z 454.598,A -85,B 0,C 180,E1 -25713.711,E2 -25713.711} C_VEL
LIN {X 0,Y 183.167,Z 446.985,A -85,B 0,C 180,E1 -25716.745,E2 -25716.745} C_VEL
LIN {X 0,Y 180.967,Z 442.168,A -85,B 0,C 180,E1 -25719.216,E2 -25719.216} C_VEL
LIN {X 0,Y 178.475,Z 437.967,A -85,B 0,C 180,E1 -25722.38,E2 -25722.38} C_VEL
LIN {X 0,Y 176.529,Z 434.556,A -85,B 0,C 180,E1 -25725.5,E2 -25725.5} C_VEL
LIN {X 0,Y 174.571,Z 431.057,A -85,B 0,C 180,E1 -25729.911,E2 -25729.911} C_VEL
LIN {X 0,Y 174.323,Z 430.47,A -85,B 0,C 180,E1 -25730.72,E2 -25730.72} C_VEL
LIN {X 0,Y 173.164,Z 429.254,A -85,B 0,C 180,E1 -25737.675,E2 -25737.675} C_VEL
LIN {X 0,Y 173.423,Z 429.486,A -85,B 0,C 180,E1 -25740.994,E2 -25740.994} C_VEL
LIN {X 0,Y 174.529,Z 430.785,A -85,B 0,C 180,E1 -25745.344,E2 -25745.344} C_VEL
LIN {X 0,Y 176.26,Z 434.247,A -85,B 0,C 180,E1 -25749.467,E2 -25749.467} C_VEL
LIN {X 0,Y 177.109,Z 435.603,A -85,B 0,C 180,E1 -25750.956,E2 -25750.956} C_VEL
LIN {X 0,Y 179.505,Z 439.752,A -85,B 0,C 180,E1 -25754.454,E2 -25754.454} C_VEL
LIN {X 0,Y 181.891,Z 443.914,A -85,B 0,C 180,E1 -25757.271,E2 -25757.271} C_VEL
LIN {X 0,Y 184.77,Z 449.144,A -85,B 0,C 180,E1 -25760.165,E2 -25760.165} C_VEL
LIN {X 0,Y 188.438,Z 456.482,A -85,B 0,C 180,E1 -25763.355,E2 -25763.355} C_VEL
LIN {X 0,Y 189.898,Z 459.664,A -85,B 0,C 180,E1 -25764.516,E2 -25764.516} C_VEL
LIN {X 0,Y 186.705,Z 492.875,A -85,B 0,C 180,E1 -25765.498,E2 -25765.498} C_VEL
LIN {X 0,Y 184.113,Z 507.389,A -85,B 0,C 180,E1 -25766.195,E2 -25766.195} C_VEL
LIN {X 0,Y 180.622,Z 520.783,A -85,B 0,C 180,E1 -25767.117,E2 -25767.117} C_VEL
LIN {X 0,Y 175.754,Z 534.671,A -85,B 0,C 180,E1 -25768.389,E2 -25768.389} C_VEL
LIN {X 0,Y 170.954,Z 545.839,A -85,B 0,C 180,E1 -25769.793,E2 -25769.793} C_VEL
LIN {X 0,Y 165.175,Z 557.255,A -85,B 0,C 180,E1 -25771.681,E2 -25771.681} C_VEL
LIN {X 0,Y 158.738,Z 567.86,A -85,B 0,C 180,E1 -25773.886,E2 -25773.886} C_VEL
LIN {X 0,Y 151.523,Z 578.37,A -85,B 0,C 180,E1 -25776.86,E2 -25776.86} C_VEL
LIN {X 0,Y 144.775,Z 587.016,A -85,B 0,C 180,E1 -25780.13,E2 -25780.13} C_VEL
LIN {X 0,Y 137.351,Z 595.268,A -85,B 0,C 180,E1 -25784.245,E2 -25784.245} C_VEL
LIN {X 0,Y 130.802,Z 601.83,A -85,B 0,C 180,E1 -25788.785,E2 -25788.785} C_VEL
LIN {X 0,Y 125.069,Z 607.089,A -85,B 0,C 180,E1 -25793.841,E2 -25793.841} C_VEL
LIN {X 0,Y 120.97,Z 610.551,A -85,B 0,C 180,E1 -25798.474,E2 -25798.474} C_VEL
LIN {X 0,Y 116.711,Z 613.883,A -85,B 0,C 180,E1 -25805.069,E2 -25805.069} C_VEL
LIN {X 0,Y 113.768,Z 615.808,A -85,B 0,C 180,E1 -25812.008,E2 -25812.008} C_VEL
LIN {X 0,Y 112.378,Z 616.375,A -85,B 0,C 180,E1 -25819.186,E2 -25819.186} C_VEL
LIN {X 0,Y 112.159,Z 615.621,A -85,B 0,C 180,E1 -25826.407,E2 -25826.407} C_VEL
LIN {X 0,Y 112.738,Z 613.557,A -85,B 0,C 180,E1 -25833.574,E2 -25833.574} C_VEL
LIN {X 0,Y 114.453,Z 610.129,A -85,B 0,C 180,E1 -25840.615,E2 -25840.615} C_VEL
LIN {X 0,Y 117.673,Z 605.22,A -85,B 0,C 180,E1 -25847.375,E2 -25847.375} C_VEL
LIN {X 0,Y 121.938,Z 598.696,A -85,B 0,C 180,E1 -25853.794,E2 -25853.794} C_VEL
LIN {X 0,Y 126.674,Z 591.442,A -85,B 0,C 180,E1 -25859.043,E2 -25859.043} C_VEL
LIN {X 0,Y 132.686,Z 582.401,A -85,B 0,C 180,E1 -25863.791,E2 -25863.791} C_VEL
LIN {X 0,Y 138.225,Z 572.96,A -85,B 0,C 180,E1 -25867.599,E2 -25867.599} C_VEL
LIN {X 0,Y 143.703,Z 562.51,A -85,B 0,C 180,E1 -25870.853,E2 -25870.853} C_VEL
LIN {X 0,Y 147.992,Z 553.514,A -85,B 0,C 180,E1 -25873.052,E2 -25873.052} C_VEL
LIN {X 0,Y 153.119,Z 541.256,A -85,B 0,C 180,E1 -25875.352,E2 -25875.352} C_VEL
LIN {X 0,Y 157.211,Z 529.491,A -85,B 0,C 180,E1 -25877.057,E2 -25877.057} C_VEL
LIN {X 0,Y 160.821,Z 516.666,A -85,B 0,C 180,E1 -25878.45,E2 -25878.45} C_VEL
LIN {X 0,Y 163.807,Z 502.065,A -85,B 0,C 180,E1 -25879.601,E2 -25879.601} C_VEL
LIN {X 0,Y 165.799,Z 487.073,A -85,B 0,C 180,E1 -25880.348,E2 -25880.348} C_VEL
LIN {X 0,Y 169.476,Z 443.096,A -85,B 0,C 180,E1 -25881.79,E2 -25881.79} C_VEL
LIN {X 0,Y 169.047,Z 441.619,A -85,B 0,C 180,E1 -25882.101,E2 -25882.101} C_VEL
LIN {X 0,Y 164.443,Z 432.154,A -85,B 0,C 180,E1 -25885.209,E2 -25885.209} C_VEL
LIN {X 0,Y 159.942,Z 424.054,A -85,B 0,C 180,E1 -25888.625,E2 -25888.625} C_VEL
LIN {X 0,Y 155.858,Z 417.264,A -85,B 0,C 180,E1 -25892.227,E2 -25892.227} C_VEL
LIN {X 0,Y 153.234,Z 413.29,A -85,B 0,C 180,E1 -25894.896,E2 -25894.896} C_VEL
LIN {X 0,Y 150.624,Z 409.407,A -85,B 0,C 180,E1 -25897.992,E2 -25897.992} C_VEL
LIN {X 0,Y 148.193,Z 405.868,A -85,B 0,C 180,E1 -25901.497,E2 -25901.497} C_VEL
LIN {X 0,Y 147.619,Z 405.021,A -85,B 0,C 180,E1 -25902.463,E2 -25902.463} C_VEL
LIN {X 0,Y 145.331,Z 402.21,A -85,B 0,C 180,E1 -25907.124,E2 -25907.124} C_VEL
LIN {X 0,Y 144.623,Z 400.149,A -85,B 0,C 180,E1 -25909.543,E2 -25909.543} C_VEL
LIN {X 0,Y 143.56,Z 399.279,A -85,B 0,C 180,E1 -25919.999,E2 -25919.999} C_VEL
LIN {X 0,Y 144.912,Z 400.474,A -85,B 0,C 180,E1 -25926.002,E2 -25926.002} C_VEL
LIN {X 0,Y 146.51,Z 403.862,A -85,B 0,C 180,E1 -25930.188,E2 -25930.188} C_VEL
LIN {X 0,Y 148.172,Z 405.608,A -85,B 0,C 180,E1 -25933.065,E2 -25933.065} C_VEL
LIN {X 0,Y 150.775,Z 409.523,A -85,B 0,C 180,E1 -25936.828,E2 -25936.828} C_VEL
LIN {X 0,Y 154.279,Z 414.858,A -85,B 0,C 180,E1 -25940.847,E2 -25940.847} C_VEL
LIN {X 0,Y 157.179,Z 419.417,A -85,B 0,C 180,E1 -25943.641,E2 -25943.641} C_VEL
LIN {X 0,Y 161.116,Z 425.997,A -85,B 0,C 180,E1 -25946.942,E2 -25946.942} C_VEL
LIN {X 0,Y 163.786,Z 432.028,A -85,B 0,C 180,E1 -25949.05,E2 -25949.05} C_VEL
LIN {X 0,Y 167.707,Z 442.441,A -85,B 0,C 180,E1 -25951.942,E2 -25951.942} C_VEL
LIN {X 0,Y 169.21,Z 447.07,A -85,B 0,C 180,E1 -25953.007,E2 -25953.007} C_VEL
LIN {X 0,Y 164.943,Z 497.567,A -85,B 0,C 180,E1 -25954.72,E2 -25954.72} C_VEL
LIN {X 0,Y 162.626,Z 511.639,A -85,B 0,C 180,E1 -25955.477,E2 -25955.477} C_VEL
LIN {X 0,Y 159.247,Z 525.749,A -85,B 0,C 180,E1 -25956.614,E2 -25956.614} C_VEL
LIN {X 0,Y 155.205,Z 538.839,A -85,B 0,C 180,E1 -25958.115,E2 -25958.115} C_VEL
LIN {X 0,Y 150.364,Z 551.51,A -85,B 0,C 180,E1 -25960.06,E2 -25960.06} C_VEL
LIN {X 0,Y 145.237,Z 563.071,A -85,B 0,C 180,E1 -25962.443,E2 -25962.443} C_VEL
LIN {X 0,Y 139.855,Z 573.674,A -85,B 0,C 180,E1 -25965.289,E2 -25965.289} C_VEL
LIN {X 0,Y 133.814,Z 584.197,A -85,B 0,C 180,E1 -25968.966,E2 -25968.966} C_VEL
LIN {X 0,Y 128.383,Z 592.876,A -85,B 0,C 180,E1 -25972.975,E2 -25972.975} C_VEL
LIN {X 0,Y 122.96,Z 601.183,A -85,B 0,C 180,E1 -25978.082,E2 -25978.082} C_VEL
LIN {X 0,Y 118.719,Z 607.867,A -85,B 0,C 180,E1 -25983.641,E2 -25983.641} C_VEL
LIN {X 0,Y 115.055,Z 613.788,A -85,B 0,C 180,E1 -25990.369,E2 -25990.369} C_VEL
LIN {X 0,Y 113.306,Z 617.209,A -85,B 0,C 180,E1 -25995.635,E2 -25995.635} C_VEL
LIN {X 0,Y 112.234,Z 620.416,A -85,B 0,C 180,E1 -26002.806,E2 -26002.806} C_VEL
LIN {X 0,Y 112.248,Z 622.221,A -85,B 0,C 180,E1 -26010,E2 -26010} C_VEL
LIN {X 0,Y 112.238,Z 622.645,A -85,B 0,C 180,E1 -26017.194,E2 -26017.194} C_VEL
LIN {X 0,Y 113.397,Z 621.742,A -85,B 0,C 180,E1 -26024.354,E2 -26024.354} C_VEL
LIN {X 0,Y 113.761,Z 621.381,A -85,B 0,C 180,E1 -26025.702,E2 -26025.702} C_VEL
LIN {X 0,Y 114.12,Z 620.575,A -85,B 0,C 180,E1 -26028.636,E2 -26028.636} C_VEL
LIN {X 0,Y 113.6,Z 618.767,A -85,B 0,C 180,E1 -26033.538,E2 -26033.538} C_VEL
LIN {X 0,Y 113.578,Z 616.96,A -85,B 0,C 180,E1 -26037.45,E2 -26037.45} C_VEL
LIN {X 0,Y 114.589,Z 615.312,A -85,B 0,C 180,E1 -26040.27,E2 -26040.27} C_VEL
LIN {X 0,Y 115.217,Z 614.69,A -85,B 0,C 180,E1 -26041.159,E2 -26041.159} C_VEL
LIN {X 0,Y 119.965,Z 610.713,A -85,B 0,C 180,E1 -26045.863,E2 -26045.863} C_VEL
LIN {X 0,Y 127.356,Z 604.015,A -85,B 0,C 180,E1 -26051.469,E2 -26051.469} C_VEL
LIN {X 0,Y 134.744,Z 596.568,A -85,B 0,C 180,E1 -26055.822,E2 -26055.822} C_VEL
LIN {X 0,Y 141.728,Z 588.807,A -85,B 0,C 180,E1 -26059.132,E2 -26059.132} C_VEL
LIN {X 0,Y 148.875,Z 579.659,A -85,B 0,C 180,E1 -26062.143,E2 -26062.143} C_VEL
LIN {X 0,Y 156.04,Z 569.192,A -85,B 0,C 180,E1 -26064.721,E2 -26064.721} C_VEL
LIN {X 0,Y 162.767,Z 557.856,A -85,B 0,C 180,E1 -26066.781,E2 -26066.781} C_VEL
LIN {X 0,Y 168.303,Z 546.908,A -85,B 0,C 180,E1 -26068.302,E2 -26068.302} C_VEL
LIN {X 0,Y 173.256,Z 535.186,A -85,B 0,C 180,E1 -26069.542,E2 -26069.542} C_VEL
LIN {X 0,Y 177.554,Z 522.473,A -85,B 0,C 180,E1 -26070.554,E2 -26070.554} C_VEL
LIN {X 0,Y 181.209,Z 507.906,A -85,B 0,C 180,E1 -26071.371,E2 -26071.371} C_VEL
LIN {X 0,Y 183.521,Z 493.875,A -85,B 0,C 180,E1 -26071.898,E2 -26071.898} C_VEL
LIN {X 0,Y 186.121,Z 466.815,A -85,B 0,C 180,E1 -26072.668,E2 -26072.668} C_VEL
LIN {X 0,Y 183.342,Z 458.772,A -85,B 0,C 180,E1 -26075.384,E2 -26075.384} C_VEL
LIN {X 0,Y 180.585,Z 451.476,A -85,B 0,C 180,E1 -26078.453,E2 -26078.453} C_VEL
LIN {X 0,Y 178.983,Z 448.032,A -85,B 0,C 180,E1 -26080.42,E2 -26080.42} C_VEL
LIN {X 0,Y 176.973,Z 444.468,A -85,B 0,C 180,E1 -26083.193,E2 -26083.193} C_VEL
LIN {X 0,Y 175.299,Z 441.336,A -85,B 0,C 180,E1 -26086.082,E2 -26086.082} C_VEL
LIN {X 0,Y 173.448,Z 437.678,A -85,B 0,C 180,E1 -26090.673,E2 -26090.673} C_VEL
LIN {X 0,Y 172.316,Z 436.489,A -85,B 0,C 180,E1 -26096.493,E2 -26096.493} C_VEL
LIN {X 0,Y 172.498,Z 436.455,A -85,B 0,C 180,E1 -26100.584,E2 -26100.584} C_VEL
LIN {X 0,Y 173.505,Z 437.754,A -85,B 0,C 180,E1 -26104.939,E2 -26104.939} C_VEL
LIN {X 0,Y 175.232,Z 441.257,A -85,B 0,C 180,E1 -26109.232,E2 -26109.232} C_VEL
LIN {X 0,Y 177.818,Z 445.937,A -85,B 0,C 180,E1 -26113.473,E2 -26113.473} C_VEL
LIN {X 0,Y 180.197,Z 450.381,A -85,B 0,C 180,E1 -26116.499,E2 -26116.499} C_VEL
LIN {X 0,Y 182.919,Z 455.655,A -85,B 0,C 180,E1 -26119.408,E2 -26119.408} C_VEL
LIN {X 0,Y 186.07,Z 462.28,A -85,B 0,C 180,E1 -26122.329,E2 -26122.329} C_VEL
LIN {X 0,Y 186.42,Z 463.112,A -85,B 0,C 180,E1 -26122.636,E2 -26122.636} C_VEL
LIN {X 0,Y 183.405,Z 493.559,A -85,B 0,C 180,E1 -26123.567,E2 -26123.567} C_VEL
LIN {X 0,Y 180.693,Z 508.056,A -85,B 0,C 180,E1 -26124.249,E2 -26124.249} C_VEL
LIN {X 0,Y 176.751,Z 522.429,A -85,B 0,C 180,E1 -26125.231,E2 -26125.231} C_VEL
LIN {X 0,Y 171.845,Z 535.77,A -85,B 0,C 180,E1 -26126.453,E2 -26126.453} C_VEL
LIN {X 0,Y 166.903,Z 546.772,A -85,B 0,C 180,E1 -26127.837,E2 -26127.837} C_VEL
LIN {X 0,Y 160.859,Z 558.206,A -85,B 0,C 180,E1 -26129.732,E2 -26129.732} C_VEL
LIN {X 0,Y 153.565,Z 569.66,A -85,B 0,C 180,E1 -26132.148,E2 -26132.148} C_VEL
LIN {X 0,Y 146.103,Z 579.847,A -85,B 0,C 180,E1 -26135.139,E2 -26135.139} C_VEL
LIN {X 0,Y 139.09,Z 588.273,A -85,B 0,C 180,E1 -26138.446,E2 -26138.446} C_VEL
LIN {X 0,Y 132.424,Z 595.282,A -85,B 0,C 180,E1 -26142.011,E2 -26142.011} C_VEL
LIN {X 0,Y 124.999,Z 602.289,A -85,B 0,C 180,E1 -26146.965,E2 -26146.965} C_VEL
LIN {X 0,Y 119.322,Z 607.179,A -85,B 0,C 180,E1 -26151.797,E2 -26151.797} C_VEL
LIN {X 0,Y 114.882,Z 610.657,A -85,B 0,C 180,E1 -26156.593,E2 -26156.593} C_VEL
LIN {X 0,Y 110.238,Z 614.02,A -85,B 0,C 180,E1 -26163.495,E2 -26163.495} C_VEL
